LIN {X 0,Y 381.733,Z 858.539,A -85,B 0,C 180,E1 -11971.054,E2 -11971.054} C_VEL
LIN {X 0,Y 381.687,Z 857.929,A -85,B 0,C 180,E1 -11972.11,E2 -11972.11} C_VEL
LIN {X 0,Y 381.699,Z 855.51,A -85,B 0,C 180,E1 -11974.223,E2 -11974.223} C_VEL
LIN {X 0,Y 381.737,Z 852.426,A -85,B 0,C 180,E1 -11975.86,E2 -11975.86} C_VEL
LIN {X 0,Y 381.947,Z 848.497,A -85,B 0,C 180,E1 -11977.4,E2 -11977.4} C_VEL
LIN {X 0,Y 382.362,Z 842.256,A -85,B 0,C 180,E1 -11979.254,E2 -11979.254} C_VEL
LIN {X 0,Y 382.84,Z 835.448,A -85,B 0,C 180,E1 -11980.845,E2 -11980.845} C_VEL
LIN {X 0,Y 383.472,Z 828.515,A -85,B 0,C 180,E1 -11982.166,E2 -11982.166} C_VEL
LIN {X 0,Y 384.235,Z 820.166,A -85,B 0,C 180,E1 -11983.485,E2 -11983.485} C_VEL
LIN {X 0,Y 384.98,Z 811.335,A -85,B 0,C 180,E1 -11984.637,E2 -11984.637} C_VEL
LIN {X 0,Y 385.832,Z 801.143,A -85,B 0,C 180,E1 -11985.72,E2 -11985.72} C_VEL
LIN {X 0,Y 386.894,Z 788.721,A -85,B 0,C 180,E1 -11986.76,E2 -11986.76} C_VEL
LIN {X 0,Y 387.324,Z 779.513,A -85,B 0,C 180,E1 -11987.375,E2 -11987.375} C_VEL
LIN {X 0,Y 386.536,Z 767.148,A -85,B 0,C 180,E1 -11988.079,E2 -11988.079} C_VEL
LIN {X 0,Y 385.447,Z 753.763,A -85,B 0,C 180,E1 -11988.616,E2 -11988.616} C_VEL
LIN {X 0,Y 383.096,Z 737.702,A -85,B 0,C 180,E1 -11989.163,E2 -11989.163} C_VEL
LIN {X 0,Y 382.769,Z 734.559,A -85,B 0,C 180,E1 -11989.403,E2 -11989.403} C_VEL
LIN {X 0,Y 383.388,Z 721.586,A -85,B 0,C 180,E1 -11993.123,E2 -11993.123} C_VEL
LIN {X 0,Y 384.077,Z 710.72,A -85,B 0,C 180,E1 -11996.282,E2 -11996.282} C_VEL
LIN {X 0,Y 385.033,Z 697.753,A -85,B 0,C 180,E1 -12000.129,E2 -12000.129} C_VEL
LIN {X 0,Y 385.892,Z 687.901,A -85,B 0,C 180,E1 -12003.117,E2 -12003.117} C_VEL
LIN {X 0,Y 386.854,Z 678.017,A -85,B 0,C 180,E1 -12006.186,E2 -12006.186} C_VEL
LIN {X 0,Y 387.104,Z 673.941,A -85,B 0,C 180,E1 -12007.489,E2 -12007.489} C_VEL
LIN {X 0,Y 385.464,Z 664.856,A -85,B 0,C 180,E1 -12010.637,E2 -12010.637} C_VEL
LIN {X 0,Y 383.783,Z 656.694,A -85,B 0,C 180,E1 -12013.623,E2 -12013.623} C_VEL
LIN {X 0,Y 383.034,Z 652.774,A -85,B 0,C 180,E1 -12015.138,E2 -12015.138} C_VEL
LIN {X 0,Y 383.072,Z 652.769,A -85,B 0,C 180,E1 -12017.248,E2 -12017.248} C_VEL
LIN {X 0,Y 383.02,Z 652.776,A -85,B 0,C 180,E1 -12020.411,E2 -12020.411} C_VEL
LIN {X 0,Y 383.023,Z 652.777,A -85,B 0,C 180,E1 -12024.044,E2 -12024.044} C_VEL
LIN {X 0,Y 382.984,Z 652.778,A -85,B 0,C 180,E1 -12027.577,E2 -12027.577} C_VEL
LIN {X 0,Y 382.993,Z 652.776,A -85,B 0,C 180,E1 -12030.3,E2 -12030.3} C_VEL
LIN {X 0,Y 383.052,Z 652.77,A -85,B 0,C 180,E1 -12032.698,E2 -12032.698} C_VEL
LIN {X 0,Y 383.048,Z 652.767,A -85,B 0,C 180,E1 -12035.039,E2 -12035.039} C_VEL
LIN {X 0,Y 382.988,Z 652.778,A -85,B 0,C 180,E1 -12038.469,E2 -12038.469} C_VEL
LIN {X 0,Y 383.084,Z 652.764,A -85,B 0,C 180,E1 -12041.827,E2 -12041.827} C_VEL
LIN {X 0,Y 383.107,Z 652.762,A -85,B 0,C 180,E1 -12045.118,E2 -12045.118} C_VEL
LIN {X 0,Y 383.105,Z 652.765,A -85,B 0,C 180,E1 -12048.358,E2 -12048.358} C_VEL
LIN {X 0,Y 383.298,Z 652.741,A -85,B 0,C 180,E1 -12051.933,E2 -12051.933} C_VEL
LIN {X 0,Y 383.194,Z 652.754,A -85,B 0,C 180,E1 -12054.738,E2 -12054.738} C_VEL
LIN {X 0,Y 383.333,Z 652.738,A -85,B 0,C 180,E1 -12058.555,E2 -12058.555} C_VEL
LIN {X 0,Y 384.693,Z 658.546,A -85,B 0,C 180,E1 -12060.523,E2 -12060.523} C_VEL
LIN {X 0,Y 386.067,Z 666.754,A -85,B 0,C 180,E1 -12063.13,E2 -12063.13} C_VEL
LIN {X 0,Y 386.301,Z 673.618,A -85,B 0,C 180,E1 -12065.219,E2 -12065.219} C_VEL
LIN {X 0,Y 385.941,Z 682.388,A -85,B 0,C 180,E1 -12067.85,E2 -12067.85} C_VEL
LIN {X 0,Y 385.494,Z 692.988,A -85,B 0,C 180,E1 -12071.036,E2 -12071.036} C_VEL
LIN {X 0,Y 384.926,Z 705.565,A -85,B 0,C 180,E1 -12074.81,E2 -12074.81} C_VEL
LIN {X 0,Y 384.421,Z 716.408,A -85,B 0,C 180,E1 -12078.107,E2 -12078.107} C_VEL
LIN {X 0,Y 383.897,Z 728.338,A -85,B 0,C 180,E1 -12081.76,E2 -12081.76} C_VEL
LIN {X 0,Y 383.867,Z 728.923,A -85,B 0,C 180,E1 -12081.938,E2 -12081.938} C_VEL
LIN {X 0,Y 386.955,Z 743.243,A -85,B 0,C 180,E1 -12082.597,E2 -12082.597} C_VEL
LIN {X 0,Y 388.559,Z 754.403,A -85,B 0,C 180,E1 -12083.237,E2 -12083.237} C_VEL
LIN {X 0,Y 387.696,Z 767.572,A -85,B 0,C 180,E1 -12084.071,E2 -12084.071} C_VEL
LIN {X 0,Y 386.831,Z 778.255,A -85,B 0,C 180,E1 -12084.958,E2 -12084.958} C_VEL
LIN {X 0,Y 385.801,Z 789.749,A -85,B 0,C 180,E1 -12086.167,E2 -12086.167} C_VEL
LIN {X 0,Y 384.839,Z 799.637,A -85,B 0,C 180,E1 -12087.459,E2 -12087.459} C_VEL
LIN {X 0,Y 384.031,Z 807.845,A -85,B 0,C 180,E1 -12088.783,E2 -12088.783} C_VEL
LIN {X 0,Y 383.205,Z 816.257,A -85,B 0,C 180,E1 -12090.462,E2 -12090.462} C_VEL
LIN {X 0,Y 382.638,Z 823.079,A -85,B 0,C 180,E1 -12092.185,E2 -12092.185} C_VEL
LIN {X 0,Y 382.072,Z 828.954,A -85,B 0,C 180,E1 -12094.133,E2 -12094.133} C_VEL
LIN {X 0,Y 381.71,Z 833.209,A -85,B 0,C 180,E1 -12096.099,E2 -12096.099} C_VEL
LIN {X 0,Y 381.529,Z 835.452,A -85,B 0,C 180,E1 -12097.621,E2 -12097.621} C_VEL
LIN {X 0,Y 381.396,Z 836.916,A -85,B 0,C 180,E1 -12099.293,E2 -12099.293} C_VEL
LIN {X 0,Y 381.312,Z 837.371,A -85,B 0,C 180,E1 -12100.917,E2 -12100.917} C_VEL
LIN {X 0,Y 381.326,Z 836.543,A -85,B 0,C 180,E1 -12102.994,E2 -12102.994} C_VEL
LIN {X 0,Y 381.455,Z 835.07,A -85,B 0,C 180,E1 -12104.436,E2 -12104.436} C_VEL
LIN {X 0,Y 381.636,Z 832.771,A -85,B 0,C 180,E1 -12105.906,E2 -12105.906} C_VEL
LIN {X 0,Y 381.904,Z 829.532,A -85,B 0,C 180,E1 -12107.4,E2 -12107.4} C_VEL
LIN {X 0,Y 382.187,Z 825.206,A -85,B 0,C 180,E1 -12108.933,E2 -12108.933} C_VEL
LIN {X 0,Y 382.644,Z 819.682,A -85,B 0,C 180,E1 -12110.481,E2 -12110.481} C_VEL
LIN {X 0,Y 383.262,Z 812.689,A -85,B 0,C 180,E1 -12112.046,E2 -12112.046} C_VEL
LIN {X 0,Y 384.074,Z 803.926,A -85,B 0,C 180,E1 -12113.623,E2 -12113.623} C_VEL
LIN {X 0,Y 384.93,Z 794.235,A -85,B 0,C 180,E1 -12115.026,E2 -12115.026} C_VEL
LIN {X 0,Y 385.773,Z 783.871,A -85,B 0,C 180,E1 -12116.234,E2 -12116.234} C_VEL
LIN {X 0,Y 386.667,Z 772.826,A -85,B 0,C 180,E1 -12117.267,E2 -12117.267} C_VEL
LIN {X 0,Y 387.487,Z 761.215,A -85,B 0,C 180,E1 -12118.114,E2 -12118.114} C_VEL
LIN {X 0,Y 387.857,Z 753.357,A -85,B 0,C 180,E1 -12118.574,E2 -12118.574} C_VEL
LIN {X 0,Y 385.883,Z 740.488,A -85,B 0,C 180,E1 -12119.256,E2 -12119.256} C_VEL
LIN {X 0,Y 383.516,Z 728.322,A -85,B 0,C 180,E1 -12119.764,E2 -12119.764} C_VEL
LIN {X 0,Y 384.031,Z 718.573,A -85,B 0,C 180,E1 -12122.774,E2 -12122.774} C_VEL
LIN {X 0,Y 384.573,Z 707.203,A -85,B 0,C 180,E1 -12126.295,E2 -12126.295} C_VEL
LIN {X 0,Y 385.051,Z 696.202,A -85,B 0,C 180,E1 -12129.71,E2 -12129.71} C_VEL
LIN {X 0,Y 385.55,Z 685.478,A -85,B 0,C 180,E1 -12133.044,E2 -12133.044} C_VEL
LIN {X 0,Y 385.996,Z 675.003,A -85,B 0,C 180,E1 -12136.309,E2 -12136.309} C_VEL
LIN {X 0,Y 386.054,Z 669.909,A -85,B 0,C 180,E1 -12137.916,E2 -12137.916} C_VEL
LIN {X 0,Y 385.13,Z 662.906,A -85,B 0,C 180,E1 -12140.202,E2 -12140.202} C_VEL
LIN {X 0,Y 383.524,Z 654.044,A -85,B 0,C 180,E1 -12143.16,E2 -12143.16} C_VEL
LIN {X 0,Y 383.28,Z 652.747,A -85,B 0,C 180,E1 -12143.618,E2 -12143.618} C_VEL
LIN {X 0,Y 383.389,Z 652.732,A -85,B 0,C 180,E1 -12147.9,E2 -12147.9} C_VEL
LIN {X 0,Y 383.521,Z 652.714,A -85,B 0,C 180,E1 -12150.001,E2 -12150.001} C_VEL
LIN {X 0,Y 383.253,Z 652.747,A -85,B 0,C 180,E1 -12153.154,E2 -12153.154} C_VEL
LIN {X 0,Y 383.283,Z 652.739,A -85,B 0,C 180,E1 -12156.317,E2 -12156.317} C_VEL
LIN {X 0,Y 383.158,Z 652.755,A -85,B 0,C 180,E1 -12159.502,E2 -12159.502} C_VEL
LIN {X 0,Y 383.135,Z 652.761,A -85,B 0,C 180,E1 -12162.856,E2 -12162.856} C_VEL
LIN {X 0,Y 383.083,Z 652.768,A -85,B 0,C 180,E1 -12165.974,E2 -12165.974} C_VEL
LIN {X 0,Y 383.097,Z 652.767,A -85,B 0,C 180,E1 -12167.427,E2 -12167.427} C_VEL
LIN {X 0,Y 382.387,Z 652.857,A -85,B 0,C 180,E1 -12167.81,E2 -12167.81} C_VEL
LIN {X 0,Y 376.706,Z 653.565,A -85,B 0,C 180,E1 -12168.908,E2 -12168.908} C_VEL
LIN {X 0,Y 376.001,Z 653.65,A -85,B 0,C 180,E1 -12169.301,E2 -12169.301} C_VEL
LIN {X 0,Y 376.03,Z 653.649,A -85,B 0,C 180,E1 -12169.944,E2 -12169.944} C_VEL
LIN {X 0,Y 379.988,Z 666.978,A -85,B 0,C 180,E1 -12171.044,E2 -12171.044} C_VEL
LIN {X 0,Y 381.497,Z 672.992,A -85,B 0,C 180,E1 -12171.62,E2 -12171.62} C_VEL
LIN {X 0,Y 380.788,Z 683.919,A -85,B 0,C 180,E1 -12172.658,E2 -12172.658} C_VEL
LIN {X 0,Y 380.039,Z 694.118,A -85,B 0,C 180,E1 -12173.862,E2 -12173.862} C_VEL
LIN {X 0,Y 379.263,Z 703.439,A -85,B 0,C 180,E1 -12175.227,E2 -12175.227} C_VEL
LIN {X 0,Y 378.52,Z 711.615,A -85,B 0,C 180,E1 -12176.692,E2 -12176.692} C_VEL
LIN {X 0,Y 377.781,Z 718.994,A -85,B 0,C 180,E1 -12178.32,E2 -12178.32} C_VEL
LIN {X 0,Y 377.252,Z 724.681,A -85,B 0,C 180,E1 -12179.89,E2 -12179.89} C_VEL
LIN {X 0,Y 376.837,Z 729.243,A -85,B 0,C 180,E1 -12181.48,E2 -12181.48} C_VEL
LIN {X 0,Y 376.408,Z 733.369,A -85,B 0,C 180,E1 -12183.422,E2 -12183.422} C_VEL
LIN {X 0,Y 376.125,Z 736.147,A -85,B 0,C 180,E1 -12185.398,E2 -12185.398} C_VEL
LIN {X 0,Y 376.045,Z 737.235,A -85,B 0,C 180,E1 -12186.731,E2 -12186.731} C_VEL
LIN {X 0,Y 376.064,Z 737.75,A -85,B 0,C 180,E1 -12188.288,E2 -12188.288} C_VEL
LIN {X 0,Y 376.219,Z 737.339,A -85,B 0,C 180,E1 -12190.013,E2 -12190.013} C_VEL
LIN {X 0,Y 376.405,Z 735.988,A -85,B 0,C 180,E1 -12191.681,E2 -12191.681} C_VEL
LIN {X 0,Y 376.818,Z 733.11,A -85,B 0,C 180,E1 -12193.637,E2 -12193.637} C_VEL
LIN {X 0,Y 377.251,Z 730.106,A -85,B 0,C 180,E1 -12195.066,E2 -12195.066} C_VEL
LIN {X 0,Y 377.875,Z 725.016,A -85,B 0,C 180,E1 -12196.887,E2 -12196.887} C_VEL
LIN {X 0,Y 378.51,Z 719.748,A -85,B 0,C 180,E1 -12198.36,E2 -12198.36} C_VEL
LIN {X 0,Y 379.263,Z 713.164,A -85,B 0,C 180,E1 -12199.852,E2 -12199.852} C_VEL
LIN {X 0,Y 380.2,Z 704.709,A -85,B 0,C 180,E1 -12201.401,E2 -12201.401} C_VEL
LIN {X 0,Y 381.046,Z 696.501,A -85,B 0,C 180,E1 -12202.619,E2 -12202.619} C_VEL
LIN {X 0,Y 381.933,Z 685.637,A -85,B 0,C 180,E1 -12203.926,E2 -12203.926} C_VEL
LIN {X 0,Y 382.716,Z 675.004,A -85,B 0,C 180,E1 -12204.943,E2 -12204.943} C_VEL
LIN {X 0,Y 380.577,Z 667.189,A -85,B 0,C 180,E1 -12205.72,E2 -12205.72} C_VEL
LIN {X 0,Y 377.058,Z 656.704,A -85,B 0,C 180,E1 -12206.643,E2 -12206.643} C_VEL
LIN {X 0,Y 376.005,Z 653.65,A -85,B 0,C 180,E1 -12206.898,E2 -12206.898} C_VEL
LIN {X 0,Y 375.965,Z 653.658,A -85,B 0,C 180,E1 -12209.688,E2 -12209.688} C_VEL
LIN {X 0,Y 376.021,Z 653.643,A -85,B 0,C 180,E1 -12213.348,E2 -12213.348} C_VEL
LIN {X 0,Y 375.984,Z 653.643,A -85,B 0,C 180,E1 -12216.888,E2 -12216.888} C_VEL
LIN {X 0,Y 376.001,Z 653.649,A -85,B 0,C 180,E1 -12220.34,E2 -12220.34} C_VEL
LIN {X 0,Y 376.034,Z 653.647,A -85,B 0,C 180,E1 -12223.719,E2 -12223.719} C_VEL
LIN {X 0,Y 376.105,Z 653.635,A -85,B 0,C 180,E1 -12227.042,E2 -12227.042} C_VEL
LIN {X 0,Y 376.12,Z 653.634,A -85,B 0,C 180,E1 -12230.319,E2 -12230.319} C_VEL
LIN {X 0,Y 376.232,Z 653.612,A -85,B 0,C 180,E1 -12232.487,E2 -12232.487} C_VEL
LIN {X 0,Y 376.173,Z 653.625,A -85,B 0,C 180,E1 -12234.64,E2 -12234.64} C_VEL
LIN {X 0,Y 376.355,Z 653.6,A -85,B 0,C 180,E1 -12237.86,E2 -12237.86} C_VEL
LIN {X 0,Y 376.491,Z 653.584,A -85,B 0,C 180,E1 -12240,E2 -12240} C_VEL
LIN {X 0,Y 376.192,Z 653.622,A -85,B 0,C 180,E1 -12243.213,E2 -12243.213} C_VEL
LIN {X 0,Y 376.248,Z 653.619,A -85,B 0,C 180,E1 -12246.435,E2 -12246.435} C_VEL
LIN {X 0,Y 376.207,Z 653.616,A -85,B 0,C 180,E1 -12248.595,E2 -12248.595} C_VEL
LIN {X 0,Y 376.052,Z 653.643,A -85,B 0,C 180,E1 -12251.864,E2 -12251.864} C_VEL
LIN {X 0,Y 376.06,Z 653.639,A -85,B 0,C 180,E1 -12255.168,E2 -12255.168} C_VEL
LIN {X 0,Y 376.026,Z 653.646,A -85,B 0,C 180,E1 -12258.526,E2 -12258.526} C_VEL
LIN {X 0,Y 375.965,Z 653.653,A -85,B 0,C 180,E1 -12261.954,E2 -12261.954} C_VEL
LIN {X 0,Y 376.008,Z 653.644,A -85,B 0,C 180,E1 -12265.461,E2 -12265.461} C_VEL
LIN {X 0,Y 375.963,Z 653.654,A -85,B 0,C 180,E1 -12269.08,E2 -12269.08} C_VEL
LIN {X 0,Y 375.951,Z 653.655,A -85,B 0,C 180,E1 -12272.829,E2 -12272.829} C_VEL
LIN {X 0,Y 375.959,Z 653.656,A -85,B 0,C 180,E1 -12275.416,E2 -12275.416} C_VEL
LIN {X 0,Y 375.976,Z 653.654,A -85,B 0,C 180,E1 -12278.27,E2 -12278.27} C_VEL
LIN {X 0,Y 375.937,Z 653.659,A -85,B 0,C 180,E1 -12281.601,E2 -12281.601} C_VEL
LIN {X 0,Y 375.993,Z 653.819,A -85,B 0,C 180,E1 -12284.646,E2 -12284.646} C_VEL
LIN {X 0,Y 377.702,Z 662.116,A -85,B 0,C 180,E1 -12288.099,E2 -12288.099} C_VEL
LIN {X 0,Y 379.191,Z 669.985,A -85,B 0,C 180,E1 -12291.118,E2 -12291.118} C_VEL
LIN {X 0,Y 379.787,Z 674.451,A -85,B 0,C 180,E1 -12292.724,E2 -12292.724} C_VEL
LIN {X 0,Y 378.937,Z 683.037,A -85,B 0,C 180,E1 -12295.551,E2 -12295.551} C_VEL
LIN {X 0,Y 377.977,Z 693.317,A -85,B 0,C 180,E1 -12298.795,E2 -12298.795} C_VEL
LIN {X 0,Y 377.175,Z 704.555,A -85,B 0,C 180,E1 -12302.236,E2 -12302.236} C_VEL
LIN {X 0,Y 376.346,Z 717.964,A -85,B 0,C 180,E1 -12306.212,E2 -12306.212} C_VEL
LIN {X 0,Y 375.686,Z 732.397,A -85,B 0,C 180,E1 -12310.393,E2 -12310.393} C_VEL
LIN {X 0,Y 377.797,Z 748.756,A -85,B 0,C 180,E1 -12311.072,E2 -12311.072} C_VEL
LIN {X 0,Y 378.667,Z 760.461,A -85,B 0,C 180,E1 -12311.658,E2 -12311.658} C_VEL
LIN {X 0,Y 379.473,Z 773.4,A -85,B 0,C 180,E1 -12312.257,E2 -12312.257} C_VEL
LIN {X 0,Y 379.949,Z 782.049,A -85,B 0,C 180,E1 -12312.785,E2 -12312.785} C_VEL
LIN {X 0,Y 379.219,Z 793.186,A -85,B 0,C 180,E1 -12313.583,E2 -12313.583} C_VEL
LIN {X 0,Y 378.271,Z 804.709,A -85,B 0,C 180,E1 -12314.647,E2 -12314.647} C_VEL
LIN {X 0,Y 377.505,Z 814.451,A -85,B 0,C 180,E1 -12315.773,E2 -12315.773} C_VEL
LIN {X 0,Y 376.746,Z 823.602,A -85,B 0,C 180,E1 -12317.064,E2 -12317.064} C_VEL
LIN {X 0,Y 375.887,Z 832.783,A -85,B 0,C 180,E1 -12318.678,E2 -12318.678} C_VEL
LIN {X 0,Y 375.344,Z 840.149,A -85,B 0,C 180,E1 -12320.298,E2 -12320.298} C_VEL
LIN {X 0,Y 374.96,Z 846.031,A -85,B 0,C 180,E1 -12321.918,E2 -12321.918} C_VEL
LIN {X 0,Y 374.717,Z 851.111,A -85,B 0,C 180,E1 -12323.744,E2 -12323.744} C_VEL
LIN {X 0,Y 374.636,Z 854.998,A -85,B 0,C 180,E1 -12325.696,E2 -12325.696} C_VEL
LIN {X 0,Y 374.543,Z 856.529,A -85,B 0,C 180,E1 -12326.772,E2 -12326.772} C_VEL
LIN {X 0,Y 374.588,Z 857.595,A -85,B 0,C 180,E1 -12327.849,E2 -12327.849} C_VEL
LIN {X 0,Y 374.647,Z 858.252,A -85,B 0,C 180,E1 -12328.925,E2 -12328.925} C_VEL
LIN {X 0,Y 374.652,Z 858.511,A -85,B 0,C 180,E1 -12329.999,E2 -12329.999} C_VEL
LIN {X 0,Y 374.645,Z 858.351,A -85,B 0,C 180,E1 -12331.074,E2 -12331.074} C_VEL
LIN {X 0,Y 374.583,Z 857.749,A -85,B 0,C 180,E1 -12332.15,E2 -12332.15} C_VEL
LIN {X 0,Y 374.624,Z 855.347,A -85,B 0,C 180,E1 -12334.303,E2 -12334.303} C_VEL
LIN {X 0,Y 374.701,Z 851.678,A -85,B 0,C 180,E1 -12336.233,E2 -12336.233} C_VEL
LIN {X 0,Y 374.974,Z 846.745,A -85,B 0,C 180,E1 -12338.08,E2 -12338.08} C_VEL
LIN {X 0,Y 375.391,Z 841.125,A -85,B 0,C 180,E1 -12339.7,E2 -12339.7} C_VEL
LIN {X 0,Y 375.928,Z 834.099,A -85,B 0,C 180,E1 -12341.32,E2 -12341.32} C_VEL
LIN {X 0,Y 376.824,Z 825.308,A -85,B 0,C 180,E1 -12342.932,E2 -12342.932} C_VEL
LIN {X 0,Y 377.581,Z 816.47,A -85,B 0,C 180,E1 -12344.257,E2 -12344.257} C_VEL
LIN {X 0,Y 378.523,Z 806.455,A -85,B 0,C 180,E1 -12345.479,E2 -12345.479} C_VEL
LIN {X 0,Y 379.52,Z 795.532,A -85,B 0,C 180,E1 -12346.541,E2 -12346.541} C_VEL
LIN {X 0,Y 380.472,Z 783.686,A -85,B 0,C 180,E1 -12347.447,E2 -12347.447} C_VEL
LIN {X 0,Y 380.157,Z 774.532,A -85,B 0,C 180,E1 -12348.041,E2 -12348.041} C_VEL
LIN {X 0,Y 379.383,Z 761.031,A -85,B 0,C 180,E1 -12348.723,E2 -12348.723} C_VEL
LIN {X 0,Y 377.751,Z 746.489,A -85,B 0,C 180,E1 -12349.237,E2 -12349.237} C_VEL
LIN {X 0,Y 376.284,Z 738.142,A -85,B 0,C 180,E1 -12349.545,E2 -12349.545} C_VEL
LIN {X 0,Y 375.791,Z 732.903,A -85,B 0,C 180,E1 -12349.956,E2 -12349.956} C_VEL
LIN {X 0,Y 376.361,Z 720.97,A -85,B 0,C 180,E1 -12353.455,E2 -12353.455} C_VEL
LIN {X 0,Y 377.073,Z 710.511,A -85,B 0,C 180,E1 -12356.571,E2 -12356.571} C_VEL
LIN {X 0,Y 377.97,Z 698.756,A -85,B 0,C 180,E1 -12360.134,E2 -12360.134} C_VEL
LIN {X 0,Y 378.943,Z 688.125,A -85,B 0,C 180,E1 -12363.427,E2 -12363.427} C_VEL
LIN {X 0,Y 380.032,Z 677.442,A -85,B 0,C 180,E1 -12366.817,E2 -12366.817} C_VEL
LIN {X 0,Y 380.108,Z 675.081,A -85,B 0,C 180,E1 -12367.6,E2 -12367.6} C_VEL
LIN {X 0,Y 378.64,Z 666.825,A -85,B 0,C 180,E1 -12370.513,E2 -12370.513} C_VEL
LIN {X 0,Y 376.911,Z 658.484,A -85,B 0,C 180,E1 -12373.622,E2 -12373.622} C_VEL
LIN {X 0,Y 376.01,Z 653.649,A -85,B 0,C 180,E1 -12375.544,E2 -12375.544} C_VEL
LIN {X 0,Y 375.998,Z 653.649,A -85,B 0,C 180,E1 -12379.14,E2 -12379.14} C_VEL
LIN {X 0,Y 375.965,Z 653.651,A -85,B 0,C 180,E1 -12381.911,E2 -12381.911} C_VEL
LIN {X 0,Y 375.976,Z 653.646,A -85,B 0,C 180,E1 -12385.332,E2 -12385.332} C_VEL
LIN {X 0,Y 375.956,Z 653.649,A -85,B 0,C 180,E1 -12388.438,E2 -12388.438} C_VEL
LIN {X 0,Y 375.998,Z 653.648,A -85,B 0,C 180,E1 -12392.141,E2 -12392.141} C_VEL
LIN {X 0,Y 376.002,Z 653.643,A -85,B 0,C 180,E1 -12394.538,E2 -12394.538} C_VEL
LIN {X 0,Y 375.958,Z 653.655,A -85,B 0,C 180,E1 -12398.045,E2 -12398.045} C_VEL
LIN {X 0,Y 376.019,Z 653.647,A -85,B 0,C 180,E1 -12401.474,E2 -12401.474} C_VEL
LIN {X 0,Y 376.055,Z 653.64,A -85,B 0,C 180,E1 -12404.832,E2 -12404.832} C_VEL
LIN {X 0,Y 376.056,Z 653.642,A -85,B 0,C 180,E1 -12408.137,E2 -12408.137} C_VEL
LIN {X 0,Y 376.252,Z 653.619,A -85,B 0,C 180,E1 -12411.877,E2 -12411.877} C_VEL
LIN {X 0,Y 376.167,Z 653.629,A -85,B 0,C 180,E1 -12414.64,E2 -12414.64} C_VEL
LIN {X 0,Y 376.345,Z 653.711,A -85,B 0,C 180,E1 -12418.06,E2 -12418.06} C_VEL
LIN {X 0,Y 378.042,Z 661.077,A -85,B 0,C 180,E1 -12420.532,E2 -12420.532} C_VEL
LIN {X 0,Y 379.191,Z 667.571,A -85,B 0,C 180,E1 -12422.656,E2 -12422.656} C_VEL
LIN {X 0,Y 379.507,Z 674.423,A -85,B 0,C 180,E1 -12424.78,E2 -12424.78} C_VEL
LIN {X 0,Y 379.168,Z 683.23,A -85,B 0,C 180,E1 -12427.455,E2 -12427.455} C_VEL
LIN {X 0,Y 378.58,Z 695.681,A -85,B 0,C 180,E1 -12431.24,E2 -12431.24} C_VEL
LIN {X 0,Y 377.989,Z 707.324,A -85,B 0,C 180,E1 -12434.8,E2 -12434.8} C_VEL
LIN {X 0,Y 377.388,Z 719.19,A -85,B 0,C 180,E1 -12438.457,E2 -12438.457} C_VEL
LIN {X 0,Y 376.944,Z 729.185,A -85,B 0,C 180,E1 -12441.548,E2 -12441.548} C_VEL
LIN {X 0,Y 379.951,Z 742.477,A -85,B 0,C 180,E1 -12442.162,E2 -12442.162} C_VEL
LIN {X 0,Y 381.78,Z 754.505,A -85,B 0,C 180,E1 -12442.867,E2 -12442.867} C_VEL
LIN {X 0,Y 381.013,Z 767.435,A -85,B 0,C 180,E1 -12443.703,E2 -12443.703} C_VEL
LIN {X 0,Y 380.013,Z 779.218,A -85,B 0,C 180,E1 -12444.703,E2 -12444.703} C_VEL
LIN {X 0,Y 379.031,Z 789.726,A -85,B 0,C 180,E1 -12445.832,E2 -12445.832} C_VEL
LIN {X 0,Y 378.083,Z 798.539,A -85,B 0,C 180,E1 -12446.988,E2 -12446.988} C_VEL
LIN {X 0,Y 377.248,Z 807.146,A -85,B 0,C 180,E1 -12448.363,E2 -12448.363} C_VEL
LIN {X 0,Y 376.371,Z 815.256,A -85,B 0,C 180,E1 -12449.967,E2 -12449.967} C_VEL
LIN {X 0,Y 375.757,Z 821.813,A -85,B 0,C 180,E1 -12451.581,E2 -12451.581} C_VEL
LIN {X 0,Y 375.316,Z 826.164,A -85,B 0,C 180,E1 -12452.891,E2 -12452.891} C_VEL
LIN {X 0,Y 374.917,Z 830.276,A -85,B 0,C 180,E1 -12454.433,E2 -12454.433} C_VEL
LIN {X 0,Y 374.6,Z 833.811,A -85,B 0,C 180,E1 -12456.223,E2 -12456.223} C_VEL
LIN {X 0,Y 374.357,Z 836.427,A -85,B 0,C 180,E1 -12458.281,E2 -12458.281} C_VEL
LIN {X 0,Y 374.29,Z 837.309,A -85,B 0,C 180,E1 -12459.673,E2 -12459.673} C_VEL
LIN {X 0,Y 374.206,Z 837.512,A -85,B 0,C 180,E1 -12461.303,E2 -12461.303} C_VEL
LIN {X 0,Y 374.224,Z 836.81,A -85,B 0,C 180,E1 -12462.911,E2 -12462.911} C_VEL
LIN {X 0,Y 374.362,Z 835.238,A -85,B 0,C 180,E1 -12464.49,E2 -12464.49} C_VEL
LIN {X 0,Y 374.626,Z 831.804,A -85,B 0,C 180,E1 -12466.556,E2 -12466.556} C_VEL
LIN {X 0,Y 374.939,Z 828.152,A -85,B 0,C 180,E1 -12468.093,E2 -12468.093} C_VEL
LIN {X 0,Y 375.311,Z 823.5,A -85,B 0,C 180,E1 -12469.623,E2 -12469.623} C_VEL
LIN {X 0,Y 375.819,Z 817.737,A -85,B 0,C 180,E1 -12471.144,E2 -12471.144} C_VEL
LIN {X 0,Y 376.458,Z 810.734,A -85,B 0,C 180,E1 -12472.648,E2 -12472.648} C_VEL
LIN {X 0,Y 377.258,Z 802.586,A -85,B 0,C 180,E1 -12474.07,E2 -12474.07} C_VEL
LIN {X 0,Y 378.127,Z 792.733,A -85,B 0,C 180,E1 -12475.468,E2 -12475.468} C_VEL
LIN {X 0,Y 379.039,Z 782.436,A -85,B 0,C 180,E1 -12476.652,E2 -12476.652} C_VEL
LIN {X 0,Y 379.956,Z 770.606,A -85,B 0,C 180,E1 -12477.727,E2 -12477.727} C_VEL
LIN {X 0,Y 380.859,Z 758.198,A -85,B 0,C 180,E1 -12478.593,E2 -12478.593} C_VEL
LIN {X 0,Y 380.867,Z 753.147,A -85,B 0,C 180,E1 -12478.892,E2 -12478.892} C_VEL
LIN {X 0,Y 378.78,Z 740.113,A -85,B 0,C 180,E1 -12479.592,E2 -12479.592} C_VEL
LIN {X 0,Y 376.548,Z 728.448,A -85,B 0,C 180,E1 -12480.088,E2 -12480.088} C_VEL
LIN {X 0,Y 377.095,Z 717.676,A -85,B 0,C 180,E1 -12483.455,E2 -12483.455} C_VEL
LIN {X 0,Y 377.673,Z 706.375,A -85,B 0,C 180,E1 -12486.998,E2 -12486.998} C_VEL
LIN {X 0,Y 378.222,Z 695.319,A -85,B 0,C 180,E1 -12490.46,E2 -12490.46} C_VEL
LIN {X 0,Y 378.823,Z 682.845,A -85,B 0,C 180,E1 -12494.382,E2 -12494.382} C_VEL
LIN {X 0,Y 379.174,Z 672.388,A -85,B 0,C 180,E1 -12497.694,E2 -12497.694} C_VEL
LIN {X 0,Y 378.504,Z 666.076,A -85,B 0,C 180,E1 -12499.767,E2 -12499.767} C_VEL
LIN {X 0,Y 376.79,Z 656.38,A -85,B 0,C 180,E1 -12503.037,E2 -12503.037} C_VEL
LIN {X 0,Y 376.225,Z 653.627,A -85,B 0,C 180,E1 -12504.036,E2 -12504.036} C_VEL
LIN {X 0,Y 376.355,Z 653.608,A -85,B 0,C 180,E1 -12507.86,E2 -12507.86} C_VEL
LIN {X 0,Y 376.49,Z 653.59,A -85,B 0,C 180,E1 -12510.001,E2 -12510.001} C_VEL
LIN {X 0,Y 376.191,Z 653.626,A -85,B 0,C 180,E1 -12513.213,E2 -12513.213} C_VEL
LIN {X 0,Y 376.241,Z 653.616,A -85,B 0,C 180,E1 -12516.436,E2 -12516.436} C_VEL
LIN {X 0,Y 376.125,Z 653.63,A -85,B 0,C 180,E1 -12519.682,E2 -12519.682} C_VEL
LIN {X 0,Y 376.091,Z 653.639,A -85,B 0,C 180,E1 -12523.658,E2 -12523.658} C_VEL
LIN {X 0,Y 376.046,Z 653.646,A -85,B 0,C 180,E1 -12527.608,E2 -12527.608} C_VEL
LIN {X 0,Y 376.001,Z 653.65,A -85,B 0,C 180,E1 -12529.301,E2 -12529.301} C_VEL
LIN {X 0,Y 375.989,Z 654.402,A -85,B 0,C 180,E1 -12529.661,E2 -12529.661} C_VEL
LIN {X 0,Y 375.944,Z 656.577,A -85,B 0,C 180,E1 -12530.015,E2 -12530.015} C_VEL
LIN {X 0,Y 375.855,Z 660.662,A -85,B 0,C 180,E1 -12530.376,E2 -12530.376} C_VEL
LIN {X 0,Y 374.837,Z 674.39,A -85,B 0,C 180,E1 -12531.373,E2 -12531.373} C_VEL
LIN {X 0,Y 374.265,Z 680.346,A -85,B 0,C 180,E1 -12531.934,E2 -12531.934} C_VEL
LIN {X 0,Y 373.485,Z 691.243,A -85,B 0,C 180,E1 -12533.137,E2 -12533.137} C_VEL
LIN {X 0,Y 372.659,Z 701.228,A -85,B 0,C 180,E1 -12534.513,E2 -12534.513} C_VEL
LIN {X 0,Y 371.821,Z 710.383,A -85,B 0,C 180,E1 -12536.07,E2 -12536.07} C_VEL
LIN {X 0,Y 371.028,Z 717.92,A -85,B 0,C 180,E1 -12537.665,E2 -12537.665} C_VEL
LIN {X 0,Y 370.347,Z 725.004,A -85,B 0,C 180,E1 -12539.565,E2 -12539.565} C_VEL
LIN {X 0,Y 369.792,Z 730.841,A -85,B 0,C 180,E1 -12541.641,E2 -12541.641} C_VEL
LIN {X 0,Y 369.384,Z 734.589,A -85,B 0,C 180,E1 -12543.488,E2 -12543.488} C_VEL
LIN {X 0,Y 369.129,Z 736.801,A -85,B 0,C 180,E1 -12545.046,E2 -12545.046} C_VEL
LIN {X 0,Y 369.012,Z 738.335,A -85,B 0,C 180,E1 -12546.879,E2 -12546.879} C_VEL
LIN {X 0,Y 369.087,Z 738.75,A -85,B 0,C 180,E1 -12548.931,E2 -12548.931} C_VEL
LIN {X 0,Y 369.236,Z 738.167,A -85,B 0,C 180,E1 -12550.416,E2 -12550.416} C_VEL
LIN {X 0,Y 369.455,Z 736.638,A -85,B 0,C 180,E1 -12552.108,E2 -12552.108} C_VEL
LIN {X 0,Y 369.86,Z 734.153,A -85,B 0,C 180,E1 -12553.775,E2 -12553.775} C_VEL
LIN {X 0,Y 370.374,Z 730.722,A -85,B 0,C 180,E1 -12555.405,E2 -12555.405} C_VEL
LIN {X 0,Y 370.956,Z 726.338,A -85,B 0,C 180,E1 -12556.997,E2 -12556.997} C_VEL
LIN {X 0,Y 371.74,Z 720.205,A -85,B 0,C 180,E1 -12558.736,E2 -12558.736} C_VEL
LIN {X 0,Y 372.549,Z 713.448,A -85,B 0,C 180,E1 -12560.264,E2 -12560.264} C_VEL
LIN {X 0,Y 373.495,Z 705.17,A -85,B 0,C 180,E1 -12561.775,E2 -12561.775} C_VEL
LIN {X 0,Y 374.43,Z 696.313,A -85,B 0,C 180,E1 -12563.085,E2 -12563.085} C_VEL
LIN {X 0,Y 375.388,Z 685.431,A -85,B 0,C 180,E1 -12564.387,E2 -12564.387} C_VEL
LIN {X 0,Y 376.04,Z 676.505,A -85,B 0,C 180,E1 -12565.249,E2 -12565.249} C_VEL
LIN {X 0,Y 373.212,Z 666.683,A -85,B 0,C 180,E1 -12566.254,E2 -12566.254} C_VEL
LIN {X 0,Y 369.027,Z 655.114,A -85,B 0,C 180,E1 -12567.279,E2 -12567.279} C_VEL
LIN {X 0,Y 368.919,Z 654.536,A -85,B 0,C 180,E1 -12567.358,E2 -12567.358} C_VEL
LIN {X 0,Y 368.916,Z 654.53,A -85,B 0,C 180,E1 -12570.31,E2 -12570.31} C_VEL
LIN {X 0,Y 369.001,Z 654.517,A -85,B 0,C 180,E1 -12574.02,E2 -12574.02} C_VEL
LIN {X 0,Y 368.926,Z 654.523,A -85,B 0,C 180,E1 -12577.605,E2 -12577.605} C_VEL
LIN {X 0,Y 368.985,Z 654.523,A -85,B 0,C 180,E1 -12581.107,E2 -12581.107} C_VEL
LIN {X 0,Y 369.002,Z 654.521,A -85,B 0,C 180,E1 -12584.536,E2 -12584.536} C_VEL
LIN {X 0,Y 369.007,Z 654.52,A -85,B 0,C 180,E1 -12587.907,E2 -12587.907} C_VEL
LIN {X 0,Y 369.231,Z 654.488,A -85,B 0,C 180,E1 -12591.801,E2 -12591.801} C_VEL
LIN {X 0,Y 369.146,Z 654.501,A -85,B 0,C 180,E1 -12594.538,E2 -12594.538} C_VEL
LIN {X 0,Y 369.32,Z 654.476,A -85,B 0,C 180,E1 -12597.819,E2 -12597.819} C_VEL
LIN {X 0,Y 369.46,Z 654.459,A -85,B 0,C 180,E1 -12600,E2 -12600} C_VEL
LIN {X 0,Y 369.321,Z 654.478,A -85,B 0,C 180,E1 -12602.181,E2 -12602.181} C_VEL
LIN {X 0,Y 369.21,Z 654.495,A -85,B 0,C 180,E1 -12606.558,E2 -12606.558} C_VEL
LIN {X 0,Y 369.139,Z 654.495,A -85,B 0,C 180,E1 -12608.761,E2 -12608.761} C_VEL
LIN {X 0,Y 369.007,Z 654.518,A -85,B 0,C 180,E1 -12612.093,E2 -12612.093} C_VEL
LIN {X 0,Y 369,Z 654.519,A -85,B 0,C 180,E1 -12615.465,E2 -12615.465} C_VEL
LIN {X 0,Y 368.984,Z 654.519,A -85,B 0,C 180,E1 -12618.893,E2 -12618.893} C_VEL
LIN {X 0,Y 368.934,Z 654.527,A -85,B 0,C 180,E1 -12622.395,E2 -12622.395} C_VEL
LIN {X 0,Y 369.002,Z 654.517,A -85,B 0,C 180,E1 -12625.98,E2 -12625.98} C_VEL
LIN {X 0,Y 368.917,Z 654.531,A -85,B 0,C 180,E1 -12629.69,E2 -12629.69} C_VEL
LIN {X 0,Y 368.899,Z 654.534,A -85,B 0,C 180,E1 -12633.043,E2 -12633.043} C_VEL
LIN {X 0,Y 368.919,Z 654.534,A -85,B 0,C 180,E1 -12636.197,E2 -12636.197} C_VEL
LIN {X 0,Y 368.905,Z 654.538,A -85,B 0,C 180,E1 -12638.953,E2 -12638.953} C_VEL
LIN {X 0,Y 368.884,Z 654.538,A -85,B 0,C 180,E1 -12642.009,E2 -12642.009} C_VEL
LIN {X 0,Y 368.961,Z 654.72,A -85,B 0,C 180,E1 -12644.161,E2 -12644.161} C_VEL
LIN {X 0,Y 370.648,Z 662.896,A -85,B 0,C 180,E1 -12647.689,E2 -12647.689} C_VEL
LIN {X 0,Y 372.117,Z 670.664,A -85,B 0,C 180,E1 -12650.746,E2 -12650.746} C_VEL
LIN {X 0,Y 372.839,Z 674.953,A -85,B 0,C 180,E1 -12652.345,E2 -12652.345} C_VEL
LIN {X 0,Y 372.147,Z 682.37,A -85,B 0,C 180,E1 -12654.866,E2 -12654.866} C_VEL
LIN {X 0,Y 371.056,Z 693.476,A -85,B 0,C 180,E1 -12658.466,E2 -12658.466} C_VEL
LIN {X 0,Y 370.114,Z 705.643,A -85,B 0,C 180,E1 -12662.275,E2 -12662.275} C_VEL
LIN {X 0,Y 369.291,Z 717.871,A -85,B 0,C 180,E1 -12665.993,E2 -12665.993} C_VEL
LIN {X 0,Y 368.643,Z 731.327,A -85,B 0,C 180,E1 -12669.985,E2 -12669.985} C_VEL
LIN {X 0,Y 370.67,Z 745.925,A -85,B 0,C 180,E1 -12670.586,E2 -12670.586} C_VEL
LIN {X 0,Y 371.895,Z 761.548,A -85,B 0,C 180,E1 -12671.39,E2 -12671.39} C_VEL
LIN {X 0,Y 372.607,Z 774.142,A -85,B 0,C 180,E1 -12672.006,E2 -12672.006} C_VEL
LIN {X 0,Y 373.068,Z 782.405,A -85,B 0,C 180,E1 -12672.528,E2 -12672.528} C_VEL
LIN {X 0,Y 372.229,Z 794.163,A -85,B 0,C 180,E1 -12673.406,E2 -12673.406} C_VEL
LIN {X 0,Y 371.274,Z 805.466,A -85,B 0,C 180,E1 -12674.491,E2 -12674.491} C_VEL
LIN {X 0,Y 370.45,Z 815.683,A -85,B 0,C 180,E1 -12675.721,E2 -12675.721} C_VEL
LIN {X 0,Y 369.639,Z 824.856,A -85,B 0,C 180,E1 -12677.09,E2 -12677.09} C_VEL
LIN {X 0,Y 368.769,Z 833.771,A -85,B 0,C 180,E1 -12678.735,E2 -12678.735} C_VEL
LIN {X 0,Y 368.222,Z 840.906,A -85,B 0,C 180,E1 -12680.386,E2 -12680.386} C_VEL
LIN {X 0,Y 367.907,Z 845.72,A -85,B 0,C 180,E1 -12681.762,E2 -12681.762} C_VEL
LIN {X 0,Y 367.65,Z 850.348,A -85,B 0,C 180,E1 -12683.413,E2 -12683.413} C_VEL
LIN {X 0,Y 367.581,Z 852.772,A -85,B 0,C 180,E1 -12684.514,E2 -12684.514} C_VEL
LIN {X 0,Y 367.562,Z 854.746,A -85,B 0,C 180,E1 -12685.613,E2 -12685.613} C_VEL
LIN {X 0,Y 367.458,Z 856.29,A -85,B 0,C 180,E1 -12686.71,E2 -12686.71} C_VEL
LIN {X 0,Y 367.486,Z 857.371,A -85,B 0,C 180,E1 -12687.807,E2 -12687.807} C_VEL
LIN {X 0,Y 367.561,Z 858.038,A -85,B 0,C 180,E1 -12688.904,E2 -12688.904} C_VEL
LIN {X 0,Y 367.584,Z 858.307,A -85,B 0,C 180,E1 -12689.999,E2 -12689.999} C_VEL
LIN {X 0,Y 367.544,Z 858.162,A -85,B 0,C 180,E1 -12691.095,E2 -12691.095} C_VEL
LIN {X 0,Y 367.48,Z 857.569,A -85,B 0,C 180,E1 -12692.191,E2 -12692.191} C_VEL
LIN {X 0,Y 367.55,Z 855.183,A -85,B 0,C 180,E1 -12694.386,E2 -12694.386} C_VEL
LIN {X 0,Y 367.595,Z 851.929,A -85,B 0,C 180,E1 -12696.182,E2 -12696.182} C_VEL
LIN {X 0,Y 367.915,Z 846.623,A -85,B 0,C 180,E1 -12698.236,E2 -12698.236} C_VEL
LIN {X 0,Y 368.368,Z 841.034,A -85,B 0,C 180,E1 -12699.887,E2 -12699.887} C_VEL
LIN {X 0,Y 368.942,Z 834.056,A -85,B 0,C 180,E1 -12701.537,E2 -12701.537} C_VEL
LIN {X 0,Y 369.896,Z 825.317,A -85,B 0,C 180,E1 -12703.179,E2 -12703.179} C_VEL
LIN {X 0,Y 370.826,Z 815.4,A -85,B 0,C 180,E1 -12704.684,E2 -12704.684} C_VEL
LIN {X 0,Y 371.803,Z 805.324,A -85,B 0,C 180,E1 -12705.907,E2 -12705.907} C_VEL
LIN {X 0,Y 372.889,Z 794.2,A -85,B 0,C 180,E1 -12706.985,E2 -12706.985} C_VEL
LIN {X 0,Y 373.812,Z 782.163,A -85,B 0,C 180,E1 -12707.904,E2 -12707.904} C_VEL
LIN {X 0,Y 373.159,Z 769.293,A -85,B 0,C 180,E1 -12708.708,E2 -12708.708} C_VEL
LIN {X 0,Y 372.202,Z 755.761,A -85,B 0,C 180,E1 -12709.33,E2 -12709.33} C_VEL
LIN {X 0,Y 370.078,Z 741.082,A -85,B 0,C 180,E1 -12709.844,E2 -12709.844} C_VEL
LIN {X 0,Y 369.507,Z 738.139,A -85,B 0,C 180,E1 -12709.967,E2 -12709.967} C_VEL
LIN {X 0,Y 368.754,Z 731.278,A -85,B 0,C 180,E1 -12710.514,E2 -12710.514} C_VEL
LIN {X 0,Y 369.395,Z 719.542,A -85,B 0,C 180,E1 -12714.043,E2 -12714.043} C_VEL
LIN {X 0,Y 370.267,Z 707.555,A -85,B 0,C 180,E1 -12717.711,E2 -12717.711} C_VEL
LIN {X 0,Y 371.348,Z 695.055,A -85,B 0,C 180,E1 -12721.608,E2 -12721.608} C_VEL
LIN {X 0,Y 372.475,Z 684.022,A -85,B 0,C 180,E1 -12725.133,E2 -12725.133} C_VEL
LIN {X 0,Y 373.078,Z 678.1,A -85,B 0,C 180,E1 -12727.07,E2 -12727.07} C_VEL
LIN {X 0,Y 372.796,Z 674.06,A -85,B 0,C 180,E1 -12728.47,E2 -12728.47} C_VEL
LIN {X 0,Y 370.991,Z 664.64,A -85,B 0,C 180,E1 -12731.92,E2 -12731.92} C_VEL
LIN {X 0,Y 368.955,Z 654.528,A -85,B 0,C 180,E1 -12735.91,E2 -12735.91} C_VEL
LIN {X 0,Y 368.95,Z 654.527,A -85,B 0,C 180,E1 -12739.635,E2 -12739.635} C_VEL
LIN {X 0,Y 368.9,Z 654.531,A -85,B 0,C 180,E1 -12743.143,E2 -12743.143} C_VEL
LIN {X 0,Y 368.893,Z 654.535,A -85,B 0,C 180,E1 -12746.461,E2 -12746.461} C_VEL
LIN {X 0,Y 368.919,Z 654.529,A -85,B 0,C 180,E1 -12750.31,E2 -12750.31} C_VEL
LIN {X 0,Y 368.977,Z 654.522,A -85,B 0,C 180,E1 -12753.534,E2 -12753.534} C_VEL
LIN {X 0,Y 368.962,Z 654.524,A -85,B 0,C 180,E1 -12756.421,E2 -12756.421} C_VEL
LIN {X 0,Y 368.931,Z 654.525,A -85,B 0,C 180,E1 -12759.947,E2 -12759.947} C_VEL
LIN {X 0,Y 368.972,Z 654.526,A -85,B 0,C 180,E1 -12763.398,E2 -12763.398} C_VEL
LIN {X 0,Y 369.055,Z 654.513,A -85,B 0,C 180,E1 -12766.79,E2 -12766.79} C_VEL
LIN {X 0,Y 369.068,Z 654.513,A -85,B 0,C 180,E1 -12770.132,E2 -12770.132} C_VEL
LIN {X 0,Y 369.183,Z 654.5,A -85,B 0,C 180,E1 -12772.342,E2 -12772.342} C_VEL
LIN {X 0,Y 369.139,Z 654.504,A -85,B 0,C 180,E1 -12774.537,E2 -12774.537} C_VEL
LIN {X 0,Y 369.235,Z 654.598,A -85,B 0,C 180,E1 -12777.409,E2 -12777.409} C_VEL
LIN {X 0,Y 371.138,Z 662.036,A -85,B 0,C 180,E1 -12780,E2 -12780} C_VEL
LIN {X 0,Y 372.508,Z 670.172,A -85,B 0,C 180,E1 -12782.703,E2 -12782.703} C_VEL
LIN {X 0,Y 372.71,Z 677.026,A -85,B 0,C 180,E1 -12784.867,E2 -12784.867} C_VEL
LIN {X 0,Y 372.29,Z 685.832,A -85,B 0,C 180,E1 -12787.593,E2 -12787.593} C_VEL
LIN {X 0,Y 371.636,Z 698.24,A -85,B 0,C 180,E1 -12791.453,E2 -12791.453} C_VEL
LIN {X 0,Y 371.09,Z 708.999,A -85,B 0,C 180,E1 -12794.751,E2 -12794.751} C_VEL
LIN {X 0,Y 370.434,Z 720.85,A -85,B 0,C 180,E1 -12798.45,E2 -12798.45} C_VEL
LIN {X 0,Y 370.039,Z 729.492,A -85,B 0,C 180,E1 -12801.116,E2 -12801.116} C_VEL
LIN {X 0,Y 373.164,Z 743.028,A -85,B 0,C 180,E1 -12801.773,E2 -12801.773} C_VEL
LIN {X 0,Y 375.126,Z 755.9,A -85,B 0,C 180,E1 -12802.568,E2 -12802.568} C_VEL
LIN {X 0,Y 374.286,Z 767.96,A -85,B 0,C 180,E1 -12803.37,E2 -12803.37} C_VEL
LIN {X 0,Y 373.302,Z 778.987,A -85,B 0,C 180,E1 -12804.32,E2 -12804.32} C_VEL
LIN {X 0,Y 372.187,Z 790.37,A -85,B 0,C 180,E1 -12805.564,E2 -12805.564} C_VEL
LIN {X 0,Y 371.104,Z 800.074,A -85,B 0,C 180,E1 -12806.881,E2 -12806.881} C_VEL
LIN {X 0,Y 370.204,Z 808.677,A -85,B 0,C 180,E1 -12808.333,E2 -12808.333} C_VEL
LIN {X 0,Y 369.297,Z 816.563,A -85,B 0,C 180,E1 -12809.971,E2 -12809.971} C_VEL
LIN {X 0,Y 368.681,Z 822.918,A -85,B 0,C 180,E1 -12811.615,E2 -12811.615} C_VEL
LIN {X 0,Y 368.042,Z 828.903,A -85,B 0,C 180,E1 -12813.626,E2 -12813.626} C_VEL
LIN {X 0,Y 367.614,Z 833.31,A -85,B 0,C 180,E1 -12815.668,E2 -12815.668} C_VEL
LIN {X 0,Y 367.318,Z 836.187,A -85,B 0,C 180,E1 -12817.753,E2 -12817.753} C_VEL
LIN {X 0,Y 367.2,Z 837.323,A -85,B 0,C 180,E1 -12819.168,E2 -12819.168} C_VEL
LIN {X 0,Y 367.146,Z 837.747,A -85,B 0,C 180,E1 -12820.605,E2 -12820.605} C_VEL
LIN {X 0,Y 367.097,Z 837.484,A -85,B 0,C 180,E1 -12822.072,E2 -12822.072} C_VEL
LIN {X 0,Y 367.173,Z 836.502,A -85,B 0,C 180,E1 -12823.556,E2 -12823.556} C_VEL
LIN {X 0,Y 367.331,Z 834.717,A -85,B 0,C 180,E1 -12825.065,E2 -12825.065} C_VEL
LIN {X 0,Y 367.563,Z 832.052,A -85,B 0,C 180,E1 -12826.6,E2 -12826.6} C_VEL
LIN {X 0,Y 367.863,Z 828.416,A -85,B 0,C 180,E1 -12828.167,E2 -12828.167} C_VEL
LIN {X 0,Y 368.318,Z 822.63,A -85,B 0,C 180,E1 -12830.07,E2 -12830.07} C_VEL
LIN {X 0,Y 369.052,Z 815.218,A -85,B 0,C 180,E1 -12831.929,E2 -12831.929} C_VEL
LIN {X 0,Y 369.76,Z 807.518,A -85,B 0,C 180,E1 -12833.475,E2 -12833.475} C_VEL
LIN {X 0,Y 370.727,Z 797.963,A -85,B 0,C 180,E1 -12835.013,E2 -12835.013} C_VEL
LIN {X 0,Y 371.757,Z 787.316,A -85,B 0,C 180,E1 -12836.392,E2 -12836.392} C_VEL
LIN {X 0,Y 372.58,Z 777.513,A -85,B 0,C 180,E1 -12837.418,E2 -12837.418} C_VEL
LIN {X 0,Y 373.53,Z 766.037,A -85,B 0,C 180,E1 -12838.368,E2 -12838.368} C_VEL
LIN {X 0,Y 374.158,Z 755.494,A -85,B 0,C 180,E1 -12839.057,E2 -12839.057} C_VEL
LIN {X 0,Y 372.179,Z 742.34,A -85,B 0,C 180,E1 -12839.817,E2 -12839.817} C_VEL
LIN {X 0,Y 369.571,Z 728.62,A -85,B 0,C 180,E1 -12840.414,E2 -12840.414} C_VEL
LIN {X 0,Y 370.238,Z 716.897,A -85,B 0,C 180,E1 -12844.114,E2 -12844.114} C_VEL
LIN {X 0,Y 370.819,Z 705.471,A -85,B 0,C 180,E1 -12847.726,E2 -12847.726} C_VEL
LIN {X 0,Y 371.358,Z 694.429,A -85,B 0,C 180,E1 -12851.233,E2 -12851.233} C_VEL
LIN {X 0,Y 371.914,Z 683.655,A -85,B 0,C 180,E1 -12854.66,E2 -12854.66} C_VEL
LIN {X 0,Y 372.264,Z 674.872,A -85,B 0,C 180,E1 -12857.461,E2 -12857.461} C_VEL
LIN {X 0,Y 371.823,Z 669.069,A -85,B 0,C 180,E1 -12859.381,E2 -12859.381} C_VEL
LIN {X 0,Y 370.346,Z 660.301,A -85,B 0,C 180,E1 -12862.367,E2 -12862.367} C_VEL
LIN {X 0,Y 369.155,Z 654.506,A -85,B 0,C 180,E1 -12864.401,E2 -12864.401} C_VEL
LIN {X 0,Y 369.32,Z 654.484,A -85,B 0,C 180,E1 -12867.819,E2 -12867.819} C_VEL
LIN {X 0,Y 369.46,Z 654.466,A -85,B 0,C 180,E1 -12870.001,E2 -12870.001} C_VEL
LIN {X 0,Y 369.32,Z 654.482,A -85,B 0,C 180,E1 -12872.182,E2 -12872.182} C_VEL
LIN {X 0,Y 369.201,Z 654.492,A -85,B 0,C 180,E1 -12876.559,E2 -12876.559} C_VEL
LIN {X 0,Y 369.124,Z 654.506,A -85,B 0,C 180,E1 -12878.762,E2 -12878.762} C_VEL
LIN {X 0,Y 369.015,Z 654.52,A -85,B 0,C 180,E1 -12882.093,E2 -12882.093} C_VEL
LIN {X 0,Y 369.001,Z 654.523,A -85,B 0,C 180,E1 -12885.465,E2 -12885.465} C_VEL
LIN {X 0,Y 368.989,Z 654.526,A -85,B 0,C 180,E1 -12888.893,E2 -12888.893} C_VEL
LIN {X 0,Y 368.983,Z 654.527,A -85,B 0,C 180,E1 -12889.616,E2 -12889.616} C_VEL
LIN {X 0,Y 372.877,Z 667.349,A -85,B 0,C 180,E1 -12890.696,E2 -12890.696} C_VEL
LIN {X 0,Y 374.578,Z 673.688,A -85,B 0,C 180,E1 -12891.317,E2 -12891.317} C_VEL
LIN {X 0,Y 374.265,Z 680.346,A -85,B 0,C 180,E1 -12891.934,E2 -12891.934} C_VEL
LIN {X 0,Y 373.287,Z 685.284,A -85,B 0,C 180,E1 -12892.409,E2 -12892.409} C_VEL
LIN {X 0,Y 369.959,Z 693.125,A -85,B 0,C 180,E1 -12893.193,E2 -12893.193} C_VEL
LIN {X 0,Y 366.595,Z 700.564,A -85,B 0,C 180,E1 -12894.072,E2 -12894.072} C_VEL
LIN {X 0,Y 365.558,Z 704.756,A -85,B 0,C 180,E1 -12894.698,E2 -12894.698} C_VEL
LIN {X 0,Y 364.674,Z 713.531,A -85,B 0,C 180,E1 -12896.312,E2 -12896.312} C_VEL
LIN {X 0,Y 363.921,Z 720.626,A -85,B 0,C 180,E1 -12897.925,E2 -12897.925} C_VEL
LIN {X 0,Y 363.256,Z 727.146,A -85,B 0,C 180,E1 -12899.798,E2 -12899.798} C_VEL
LIN {X 0,Y 362.812,Z 731.808,A -85,B 0,C 180,E1 -12901.535,E2 -12901.535} C_VEL
LIN {X 0,Y 362.353,Z 735.694,A -85,B 0,C 180,E1 -12903.488,E2 -12903.488} C_VEL
LIN {X 0,Y 362.071,Z 738.453,A -85,B 0,C 180,E1 -12905.614,E2 -12905.614} C_VEL
LIN {X 0,Y 361.994,Z 739.549,A -85,B 0,C 180,E1 -12907.25,E2 -12907.25} C_VEL
LIN {X 0,Y 362.073,Z 739.781,A -85,B 0,C 180,E1 -12909.066,E2 -12909.066} C_VEL
LIN {X 0,Y 362.324,Z 738.646,A -85,B 0,C 180,E1 -12911.262,E2 -12911.262} C_VEL
LIN {X 0,Y 362.783,Z 735.999,A -85,B 0,C 180,E1 -12913.45,E2 -12913.45} C_VEL
LIN {X 0,Y 363.216,Z 733.234,A -85,B 0,C 180,E1 -12914.93,E2 -12914.93} C_VEL
LIN {X 0,Y 363.923,Z 728.498,A -85,B 0,C 180,E1 -12916.834,E2 -12916.834} C_VEL
LIN {X 0,Y 364.756,Z 722.249,A -85,B 0,C 180,E1 -12918.716,E2 -12918.716} C_VEL
LIN {X 0,Y 365.588,Z 715.773,A -85,B 0,C 180,E1 -12920.26,E2 -12920.26} C_VEL
LIN {X 0,Y 366.665,Z 706.975,A -85,B 0,C 180,E1 -12921.948,E2 -12921.948} C_VEL
LIN {X 0,Y 367.715,Z 697.475,A -85,B 0,C 180,E1 -12923.392,E2 -12923.392} C_VEL
LIN {X 0,Y 368.636,Z 687.645,A -85,B 0,C 180,E1 -12924.602,E2 -12924.602} C_VEL
LIN {X 0,Y 369.339,Z 678.515,A -85,B 0,C 180,E1 -12925.521,E2 -12925.521} C_VEL
LIN {X 0,Y 366.709,Z 669.043,A -85,B 0,C 180,E1 -12926.527,E2 -12926.527} C_VEL
LIN {X 0,Y 362.991,Z 658.714,A -85,B 0,C 180,E1 -12927.502,E2 -12927.502} C_VEL
LIN {X 0,Y 361.87,Z 655.411,A -85,B 0,C 180,E1 -12927.8,E2 -12927.8} C_VEL
LIN {X 0,Y 361.901,Z 655.402,A -85,B 0,C 180,E1 -12930.955,E2 -12930.955} C_VEL
LIN {X 0,Y 361.955,Z 655.394,A -85,B 0,C 180,E1 -12933.475,E2 -12933.475} C_VEL
LIN {X 0,Y 361.883,Z 655.398,A -85,B 0,C 180,E1 -12937.144,E2 -12937.144} C_VEL
LIN {X 0,Y 361.923,Z 655.402,A -85,B 0,C 180,E1 -12940.724,E2 -12940.724} C_VEL
LIN {X 0,Y 361.95,Z 655.402,A -85,B 0,C 180,E1 -12944.226,E2 -12944.226} C_VEL
LIN {X 0,Y 362,Z 655.393,A -85,B 0,C 180,E1 -12946.528,E2 -12946.528} C_VEL
LIN {X 0,Y 362.033,Z 655.39,A -85,B 0,C 180,E1 -12949.938,E2 -12949.938} C_VEL
LIN {X 0,Y 362.153,Z 655.366,A -85,B 0,C 180,E1 -12952.193,E2 -12952.193} C_VEL
LIN {X 0,Y 362.12,Z 655.377,A -85,B 0,C 180,E1 -12954.431,E2 -12954.431} C_VEL
LIN {X 0,Y 362.284,Z 655.351,A -85,B 0,C 180,E1 -12957.777,E2 -12957.777} C_VEL
LIN {X 0,Y 362.43,Z 655.334,A -85,B 0,C 180,E1 -12960,E2 -12960} C_VEL
LIN {X 0,Y 362.285,Z 655.355,A -85,B 0,C 180,E1 -12962.224,E2 -12962.224} C_VEL
LIN {X 0,Y 362.174,Z 655.37,A -85,B 0,C 180,E1 -12966.686,E2 -12966.686} C_VEL
LIN {X 0,Y 362.076,Z 655.374,A -85,B 0,C 180,E1 -12968.933,E2 -12968.933} C_VEL
LIN {X 0,Y 361.962,Z 655.393,A -85,B 0,C 180,E1 -12972.332,E2 -12972.332} C_VEL
LIN {X 0,Y 361.964,Z 655.398,A -85,B 0,C 180,E1 -12974.62,E2 -12974.62} C_VEL
LIN {X 0,Y 361.962,Z 655.397,A -85,B 0,C 180,E1 -12978.099,E2 -12978.099} C_VEL
LIN {X 0,Y 361.894,Z 655.404,A -85,B 0,C 180,E1 -12981.653,E2 -12981.653} C_VEL
LIN {X 0,Y 361.93,Z 655.398,A -85,B 0,C 180,E1 -12985.29,E2 -12985.29} C_VEL
LIN {X 0,Y 361.91,Z 655.403,A -85,B 0,C 180,E1 -12987.779,E2 -12987.779} C_VEL
LIN {X 0,Y 361.84,Z 655.413,A -85,B 0,C 180,E1 -12991.629,E2 -12991.629} C_VEL
LIN {X 0,Y 361.876,Z 655.411,A -85,B 0,C 180,E1 -12995.345,E2 -12995.345} C_VEL
LIN {X 0,Y 361.872,Z 655.413,A -85,B 0,C 180,E1 -12999.027,E2 -12999.027} C_VEL
LIN {X 0,Y 361.838,Z 655.409,A -85,B 0,C 180,E1 -13002.829,E2 -13002.829} C_VEL
LIN {X 0,Y 361.861,Z 655.522,A -85,B 0,C 180,E1 -13003.603,E2 -13003.603} C_VEL
LIN {X 0,Y 363.237,Z 661.954,A -85,B 0,C 180,E1 -13006.515,E2 -13006.515} C_VEL
LIN {X 0,Y 364.81,Z 669.854,A -85,B 0,C 180,E1 -13009.777,E2 -13009.777} C_VEL
LIN {X 0,Y 365.821,Z 675.772,A -85,B 0,C 180,E1 -13012.064,E2 -13012.064} C_VEL
LIN {X 0,Y 365.663,Z 679.611,A -85,B 0,C 180,E1 -13013.429,E2 -13013.429} C_VEL
LIN {X 0,Y 364.371,Z 691.14,A -85,B 0,C 180,E1 -13017.312,E2 -13017.312} C_VEL
LIN {X 0,Y 363.302,Z 702.776,A -85,B 0,C 180,E1 -13021.078,E2 -13021.078} C_VEL
LIN {X 0,Y 362.461,Z 714.506,A -85,B 0,C 180,E1 -13024.749,E2 -13024.749} C_VEL
LIN {X 0,Y 361.717,Z 727.91,A -85,B 0,C 180,E1 -13028.847,E2 -13028.847} C_VEL
LIN {X 0,Y 361.6,Z 730.15,A -85,B 0,C 180,E1 -13029.522,E2 -13029.522} C_VEL
LIN {X 0,Y 363.848,Z 745.813,A -85,B 0,C 180,E1 -13030.207,E2 -13030.207} C_VEL
LIN {X 0,Y 365.049,Z 761.893,A -85,B 0,C 180,E1 -13031.089,E2 -13031.089} C_VEL
LIN {X 0,Y 365.763,Z 774.723,A -85,B 0,C 180,E1 -13031.74,E2 -13031.74} C_VEL
LIN {X 0,Y 366.186,Z 782.73,A -85,B 0,C 180,E1 -13032.261,E2 -13032.261} C_VEL
LIN {X 0,Y 365.415,Z 793.573,A -85,B 0,C 180,E1 -13033.088,E2 -13033.088} C_VEL
LIN {X 0,Y 364.387,Z 804.941,A -85,B 0,C 180,E1 -13034.191,E2 -13034.191} C_VEL
LIN {X 0,Y 363.517,Z 815.22,A -85,B 0,C 180,E1 -13035.443,E2 -13035.443} C_VEL
LIN {X 0,Y 362.679,Z 824.448,A -85,B 0,C 180,E1 -13036.838,E2 -13036.838} C_VEL
LIN {X 0,Y 361.767,Z 833.399,A -85,B 0,C 180,E1 -13038.514,E2 -13038.514} C_VEL
LIN {X 0,Y 361.189,Z 840.576,A -85,B 0,C 180,E1 -13040.197,E2 -13040.197} C_VEL
LIN {X 0,Y 360.735,Z 847.074,A -85,B 0,C 180,E1 -13042.161,E2 -13042.161} C_VEL
LIN {X 0,Y 360.53,Z 851.26,A -85,B 0,C 180,E1 -13043.812,E2 -13043.812} C_VEL
LIN {X 0,Y 360.468,Z 854.492,A -85,B 0,C 180,E1 -13045.527,E2 -13045.527} C_VEL
LIN {X 0,Y 360.376,Z 856.049,A -85,B 0,C 180,E1 -13046.645,E2 -13046.645} C_VEL
LIN {X 0,Y 360.384,Z 857.148,A -85,B 0,C 180,E1 -13047.764,E2 -13047.764} C_VEL
LIN {X 0,Y 360.46,Z 857.824,A -85,B 0,C 180,E1 -13048.882,E2 -13048.882} C_VEL
LIN {X 0,Y 360.498,Z 858.102,A -85,B 0,C 180,E1 -13049.999,E2 -13049.999} C_VEL
LIN {X 0,Y 360.443,Z 857.971,A -85,B 0,C 180,E1 -13051.117,E2 -13051.117} C_VEL
LIN {X 0,Y 360.378,Z 857.389,A -85,B 0,C 180,E1 -13052.235,E2 -13052.235} C_VEL
LIN {X 0,Y 360.455,Z 855.024,A -85,B 0,C 180,E1 -13054.472,E2 -13054.472} C_VEL
LIN {X 0,Y 360.492,Z 852.142,A -85,B 0,C 180,E1 -13056.132,E2 -13056.132} C_VEL
LIN {X 0,Y 360.737,Z 848.124,A -85,B 0,C 180,E1 -13057.838,E2 -13057.838} C_VEL
LIN {X 0,Y 361.238,Z 841.984,A -85,B 0,C 180,E1 -13059.801,E2 -13059.801} C_VEL
LIN {X 0,Y 361.838,Z 835.262,A -85,B 0,C 180,E1 -13061.483,E2 -13061.483} C_VEL
LIN {X 0,Y 362.809,Z 826.938,A -85,B 0,C 180,E1 -13063.156,E2 -13063.156} C_VEL
LIN {X 0,Y 363.742,Z 817.249,A -85,B 0,C 180,E1 -13064.712,E2 -13064.712} C_VEL
LIN {X 0,Y 364.852,Z 806.688,A -85,B 0,C 180,E1 -13066.075,E2 -13066.075} C_VEL
LIN {X 0,Y 365.972,Z 796.013,A -85,B 0,C 180,E1 -13067.172,E2 -13067.172} C_VEL
LIN {X 0,Y 366.992,Z 784.352,A -85,B 0,C 180,E1 -13068.117,E2 -13068.117} C_VEL
LIN {X 0,Y 366.568,Z 771.847,A -85,B 0,C 180,E1 -13068.967,E2 -13068.967} C_VEL
LIN {X 0,Y 365.806,Z 758.834,A -85,B 0,C 180,E1 -13069.619,E2 -13069.619} C_VEL
LIN {X 0,Y 364.201,Z 746.099,A -85,B 0,C 180,E1 -13070.102,E2 -13070.102} C_VEL
LIN {X 0,Y 362.715,Z 738.228,A -85,B 0,C 180,E1 -13070.411,E2 -13070.411} C_VEL
LIN {X 0,Y 361.766,Z 729.431,A -85,B 0,C 180,E1 -13071.173,E2 -13071.173} C_VEL
LIN {X 0,Y 362.627,Z 716.232,A -85,B 0,C 180,E1 -13075.237,E2 -13075.237} C_VEL
LIN {X 0,Y 363.601,Z 703.506,A -85,B 0,C 180,E1 -13079.246,E2 -13079.246} C_VEL
LIN {X 0,Y 364.848,Z 690.909,A -85,B 0,C 180,E1 -13083.297,E2 -13083.297} C_VEL
LIN {X 0,Y 365.919,Z 681.096,A -85,B 0,C 180,E1 -13086.54,E2 -13086.54} C_VEL
LIN {X 0,Y 366.036,Z 676.606,A -85,B 0,C 180,E1 -13088.074,E2 -13088.074} C_VEL
LIN {X 0,Y 364.43,Z 668.115,A -85,B 0,C 180,E1 -13091.226,E2 -13091.226} C_VEL
LIN {X 0,Y 362.514,Z 658.598,A -85,B 0,C 180,E1 -13094.958,E2 -13094.958} C_VEL
LIN {X 0,Y 361.911,Z 655.405,A -85,B 0,C 180,E1 -13096.29,E2 -13096.29} C_VEL
LIN {X 0,Y 361.878,Z 655.41,A -85,B 0,C 180,E1 -13100.141,E2 -13100.141} C_VEL
LIN {X 0,Y 361.866,Z 655.406,A -85,B 0,C 180,E1 -13102.982,E2 -13102.982} C_VEL
LIN {X 0,Y 361.855,Z 655.411,A -85,B 0,C 180,E1 -13106.63,E2 -13106.63} C_VEL
LIN {X 0,Y 361.872,Z 655.409,A -85,B 0,C 180,E1 -13109.672,E2 -13109.672} C_VEL
LIN {X 0,Y 361.95,Z 655.398,A -85,B 0,C 180,E1 -13113.475,E2 -13113.475} C_VEL
LIN {X 0,Y 361.885,Z 655.402,A -85,B 0,C 180,E1 -13117.144,E2 -13117.144} C_VEL
LIN {X 0,Y 361.916,Z 655.402,A -85,B 0,C 180,E1 -13120.724,E2 -13120.724} C_VEL
LIN {X 0,Y 361.942,Z 655.4,A -85,B 0,C 180,E1 -13124.226,E2 -13124.226} C_VEL
LIN {X 0,Y 361.995,Z 655.394,A -85,B 0,C 180,E1 -13126.527,E2 -13126.527} C_VEL
LIN {X 0,Y 362.032,Z 655.389,A -85,B 0,C 180,E1 -13129.938,E2 -13129.938} C_VEL
LIN {X 0,Y 362.146,Z 655.378,A -85,B 0,C 180,E1 -13132.192,E2 -13132.192} C_VEL
LIN {X 0,Y 362.113,Z 655.379,A -85,B 0,C 180,E1 -13134.431,E2 -13134.431} C_VEL
LIN {X 0,Y 362.12,Z 655.545,A -85,B 0,C 180,E1 -13136.732,E2 -13136.732} C_VEL
LIN {X 0,Y 363.723,Z 661.523,A -85,B 0,C 180,E1 -13138.893,E2 -13138.893} C_VEL
LIN {X 0,Y 365.058,Z 667.883,A -85,B 0,C 180,E1 -13141.103,E2 -13141.103} C_VEL
LIN {X 0,Y 365.805,Z 672.78,A -85,B 0,C 180,E1 -13142.753,E2 -13142.753} C_VEL
LIN {X 0,Y 365.913,Z 679.666,A -85,B 0,C 180,E1 -13144.958,E2 -13144.958} C_VEL
LIN {X 0,Y 365.402,Z 688.412,A -85,B 0,C 180,E1 -13147.737,E2 -13147.737} C_VEL
LIN {X 0,Y 364.851,Z 699.25,A -85,B 0,C 180,E1 -13151.106,E2 -13151.106} C_VEL
LIN {X 0,Y 364.209,Z 710.168,A -85,B 0,C 180,E1 -13154.528,E2 -13154.528} C_VEL
LIN {X 0,Y 363.573,Z 721.208,A -85,B 0,C 180,E1 -13158.016,E2 -13158.016} C_VEL
LIN {X 0,Y 363.131,Z 729.486,A -85,B 0,C 180,E1 -13160.647,E2 -13160.647} C_VEL
LIN {X 0,Y 366.338,Z 743.115,A -85,B 0,C 180,E1 -13161.34,E2 -13161.34} C_VEL
LIN {X 0,Y 368.427,Z 756.712,A -85,B 0,C 180,E1 -13162.206,E2 -13162.206} C_VEL
LIN {X 0,Y 367.6,Z 768.652,A -85,B 0,C 180,E1 -13163.029,E2 -13163.029} C_VEL
LIN {X 0,Y 366.507,Z 780.043,A -85,B 0,C 180,E1 -13164.047,E2 -13164.047} C_VEL
LIN {X 0,Y 365.341,Z 791.12,A -85,B 0,C 180,E1 -13165.296,E2 -13165.296} C_VEL
LIN {X 0,Y 364.204,Z 800.714,A -85,B 0,C 180,E1 -13166.641,E2 -13166.641} C_VEL
LIN {X 0,Y 363.149,Z 810.194,A -85,B 0,C 180,E1 -13168.304,E2 -13168.304} C_VEL
LIN {X 0,Y 362.2,Z 818.079,A -85,B 0,C 180,E1 -13170.029,E2 -13170.029} C_VEL
LIN {X 0,Y 361.495,Z 825.043,A -85,B 0,C 180,E1 -13171.991,E2 -13171.991} C_VEL
LIN {X 0,Y 360.951,Z 829.859,A -85,B 0,C 180,E1 -13173.744,E2 -13173.744} C_VEL
LIN {X 0,Y 360.515,Z 833.951,A -85,B 0,C 180,E1 -13175.791,E2 -13175.791} C_VEL
LIN {X 0,Y 360.301,Z 835.929,A -85,B 0,C 180,E1 -13177.206,E2 -13177.206} C_VEL
LIN {X 0,Y 360.13,Z 837.258,A -85,B 0,C 180,E1 -13178.685,E2 -13178.685} C_VEL
LIN {X 0,Y 360.049,Z 837.933,A -85,B 0,C 180,E1 -13180.426,E2 -13180.426} C_VEL
LIN {X 0,Y 360.018,Z 837.657,A -85,B 0,C 180,E1 -13182.116,E2 -13182.116} C_VEL
LIN {X 0,Y 360.093,Z 836.496,A -85,B 0,C 180,E1 -13183.77,E2 -13183.77} C_VEL
LIN {X 0,Y 360.287,Z 834.48,A -85,B 0,C 180,E1 -13185.394,E2 -13185.394} C_VEL
LIN {X 0,Y 360.559,Z 831.627,A -85,B 0,C 180,E1 -13186.984,E2 -13186.984} C_VEL
LIN {X 0,Y 360.952,Z 826.606,A -85,B 0,C 180,E1 -13189.001,E2 -13189.001} C_VEL
LIN {X 0,Y 361.422,Z 821.473,A -85,B 0,C 180,E1 -13190.585,E2 -13190.585} C_VEL
LIN {X 0,Y 362.073,Z 815.104,A -85,B 0,C 180,E1 -13192.172,E2 -13192.172} C_VEL
LIN {X 0,Y 362.846,Z 807.328,A -85,B 0,C 180,E1 -13193.747,E2 -13193.747} C_VEL
LIN {X 0,Y 363.784,Z 798.058,A -85,B 0,C 180,E1 -13195.257,E2 -13195.257} C_VEL
LIN {X 0,Y 364.76,Z 788.366,A -85,B 0,C 180,E1 -13196.542,E2 -13196.542} C_VEL
LIN {X 0,Y 365.73,Z 777.314,A -85,B 0,C 180,E1 -13197.728,E2 -13197.728} C_VEL
LIN {X 0,Y 366.76,Z 764.81,A -85,B 0,C 180,E1 -13198.764,E2 -13198.764} C_VEL
LIN {X 0,Y 367.215,Z 755.374,A -85,B 0,C 180,E1 -13199.384,E2 -13199.384} C_VEL
LIN {X 0,Y 365.218,Z 742.373,A -85,B 0,C 180,E1 -13200.148,E2 -13200.148} C_VEL
LIN {X 0,Y 362.632,Z 728.738,A -85,B 0,C 180,E1 -13200.757,E2 -13200.757} C_VEL
LIN {X 0,Y 363.255,Z 717.984,A -85,B 0,C 180,E1 -13204.196,E2 -13204.196} C_VEL
LIN {X 0,Y 363.872,Z 706.126,A -85,B 0,C 180,E1 -13207.986,E2 -13207.986} C_VEL
LIN {X 0,Y 364.428,Z 695.247,A -85,B 0,C 180,E1 -13211.481,E2 -13211.481} C_VEL
LIN {X 0,Y 365.008,Z 684.505,A -85,B 0,C 180,E1 -13214.935,E2 -13214.935} C_VEL
LIN {X 0,Y 365.353,Z 675.694,A -85,B 0,C 180,E1 -13217.785,E2 -13217.785} C_VEL
LIN {X 0,Y 364.683,Z 669.075,A -85,B 0,C 180,E1 -13220.013,E2 -13220.013} C_VEL
LIN {X 0,Y 363,Z 659.513,A -85,B 0,C 180,E1 -13223.33,E2 -13223.33} C_VEL
LIN {X 0,Y 362.046,Z 655.392,A -85,B 0,C 180,E1 -13224.85,E2 -13224.85} C_VEL
LIN {X 0,Y 362.284,Z 655.361,A -85,B 0,C 180,E1 -13227.777,E2 -13227.777} C_VEL
LIN {X 0,Y 362.429,Z 655.342,A -85,B 0,C 180,E1 -13230.001,E2 -13230.001} C_VEL
LIN {X 0,Y 362.284,Z 655.358,A -85,B 0,C 180,E1 -13232.224,E2 -13232.224} C_VEL
LIN {X 0,Y 362.163,Z 655.369,A -85,B 0,C 180,E1 -13236.687,E2 -13236.687} C_VEL
LIN {X 0,Y 362.037,Z 655.385,A -85,B 0,C 180,E1 -13240.062,E2 -13240.062} C_VEL
LIN {X 0,Y 362,Z 655.395,A -85,B 0,C 180,E1 -13243.9,E2 -13243.9} C_VEL
LIN {X 0,Y 361.969,Z 655.401,A -85,B 0,C 180,E1 -13247.939,E2 -13247.939} C_VEL
LIN {X 0,Y 361.947,Z 655.403,A -85,B 0,C 180,E1 -13249.275,E2 -13249.275} C_VEL
LIN {X 0,Y 365.826,Z 668.215,A -85,B 0,C 180,E1 -13250.378,E2 -13250.378} C_VEL
LIN {X 0,Y 367.837,Z 675.756,A -85,B 0,C 180,E1 -13251.139,E2 -13251.139} C_VEL
LIN {X 0,Y 367.09,Z 686.559,A -85,B 0,C 180,E1 -13252.218,E2 -13252.218} C_VEL
LIN {X 0,Y 366.229,Z 697.218,A -85,B 0,C 180,E1 -13253.553,E2 -13253.553} C_VEL
LIN {X 0,Y 365.558,Z 704.756,A -85,B 0,C 180,E1 -13254.698,E2 -13254.698} C_VEL
LIN {X 0,Y 364.526,Z 708.816,A -85,B 0,C 180,E1 -13255.352,E2 -13255.352} C_VEL
LIN {X 0,Y 361.131,Z 715.13,A -85,B 0,C 180,E1 -13256.435,E2 -13256.435} C_VEL
LIN {X 0,Y 357.747,Z 720.858,A -85,B 0,C 180,E1 -13257.609,E2 -13257.609} C_VEL
LIN {X 0,Y 356.752,Z 723.962,A -85,B 0,C 180,E1 -13258.398,E2 -13258.398} C_VEL
LIN {X 0,Y 356.089,Z 729.888,A -85,B 0,C 180,E1 -13260.272,E2 -13260.272} C_VEL
LIN {X 0,Y 355.606,Z 734.569,A -85,B 0,C 180,E1 -13262.25,E2 -13262.25} C_VEL
LIN {X 0,Y 355.272,Z 737.328,A -85,B 0,C 180,E1 -13263.814,E2 -13263.814} C_VEL
LIN {X 0,Y 355.028,Z 739.593,A -85,B 0,C 180,E1 -13265.746,E2 -13265.746} C_VEL
LIN {X 0,Y 354.973,Z 740.748,A -85,B 0,C 180,E1 -13267.862,E2 -13267.862} C_VEL
LIN {X 0,Y 355.091,Z 740.722,A -85,B 0,C 180,E1 -13269.476,E2 -13269.476} C_VEL
LIN {X 0,Y 355.316,Z 739.767,A -85,B 0,C 180,E1 -13271.269,E2 -13271.269} C_VEL
LIN {X 0,Y 355.639,Z 737.883,A -85,B 0,C 180,E1 -13273.015,E2 -13273.015} C_VEL
LIN {X 0,Y 356.327,Z 734.009,A -85,B 0,C 180,E1 -13275.239,E2 -13275.239} C_VEL
LIN {X 0,Y 356.916,Z 730.3,A -85,B 0,C 180,E1 -13276.766,E2 -13276.766} C_VEL
LIN {X 0,Y 357.729,Z 724.443,A -85,B 0,C 180,E1 -13278.658,E2 -13278.658} C_VEL
LIN {X 0,Y 358.612,Z 717.998,A -85,B 0,C 180,E1 -13280.284,E2 -13280.284} C_VEL
LIN {X 0,Y 359.6,Z 710.575,A -85,B 0,C 180,E1 -13281.796,E2 -13281.796} C_VEL
LIN {X 0,Y 360.76,Z 700.961,A -85,B 0,C 180,E1 -13283.378,E2 -13283.378} C_VEL
LIN {X 0,Y 361.791,Z 691.17,A -85,B 0,C 180,E1 -13284.674,E2 -13284.674} C_VEL
LIN {X 0,Y 362.686,Z 680.446,A -85,B 0,C 180,E1 -13285.809,E2 -13285.809} C_VEL
LIN {X 0,Y 360.453,Z 672.065,A -85,B 0,C 180,E1 -13286.745,E2 -13286.745} C_VEL
LIN {X 0,Y 357.025,Z 662.274,A -85,B 0,C 180,E1 -13287.727,E2 -13287.727} C_VEL
LIN {X 0,Y 354.817,Z 656.288,A -85,B 0,C 180,E1 -13288.263,E2 -13288.263} C_VEL
LIN {X 0,Y 354.849,Z 656.285,A -85,B 0,C 180,E1 -13291.619,E2 -13291.619} C_VEL
LIN {X 0,Y 354.9,Z 656.273,A -85,B 0,C 180,E1 -13294.173,E2 -13294.173} C_VEL
LIN {X 0,Y 354.828,Z 656.281,A -85,B 0,C 180,E1 -13297.894,E2 -13297.894} C_VEL
LIN {X 0,Y 354.925,Z 656.278,A -85,B 0,C 180,E1 -13301.891,E2 -13301.891} C_VEL
LIN {X 0,Y 354.944,Z 656.271,A -85,B 0,C 180,E1 -13305.981,E2 -13305.981} C_VEL
LIN {X 0,Y 354.979,Z 656.266,A -85,B 0,C 180,E1 -13309.736,E2 -13309.736} C_VEL
LIN {X 0,Y 355.116,Z 656.243,A -85,B 0,C 180,E1 -13312.037,E2 -13312.037} C_VEL
LIN {X 0,Y 355.094,Z 656.253,A -85,B 0,C 180,E1 -13314.321,E2 -13314.321} C_VEL
LIN {X 0,Y 355.247,Z 656.227,A -85,B 0,C 180,E1 -13317.733,E2 -13317.733} C_VEL
LIN {X 0,Y 355.399,Z 656.21,A -85,B 0,C 180,E1 -13320,E2 -13320} C_VEL
LIN {X 0,Y 355.248,Z 656.232,A -85,B 0,C 180,E1 -13322.268,E2 -13322.268} C_VEL
LIN {X 0,Y 355.14,Z 656.246,A -85,B 0,C 180,E1 -13326.819,E2 -13326.819} C_VEL
LIN {X 0,Y 355.017,Z 656.253,A -85,B 0,C 180,E1 -13329.112,E2 -13329.112} C_VEL
LIN {X 0,Y 354.923,Z 656.268,A -85,B 0,C 180,E1 -13332.581,E2 -13332.581} C_VEL
LIN {X 0,Y 354.891,Z 656.275,A -85,B 0,C 180,E1 -13336.096,E2 -13336.096} C_VEL
LIN {X 0,Y 354.908,Z 656.277,A -85,B 0,C 180,E1 -13338.472,E2 -13338.472} C_VEL
LIN {X 0,Y 354.837,Z 656.286,A -85,B 0,C 180,E1 -13342.106,E2 -13342.106} C_VEL
LIN {X 0,Y 354.901,Z 656.273,A -85,B 0,C 180,E1 -13345.827,E2 -13345.827} C_VEL
LIN {X 0,Y 354.82,Z 656.287,A -85,B 0,C 180,E1 -13349.682,E2 -13349.682} C_VEL
LIN {X 0,Y 354.808,Z 656.29,A -85,B 0,C 180,E1 -13353.702,E2 -13353.702} C_VEL
LIN {X 0,Y 354.8,Z 656.292,A -85,B 0,C 180,E1 -13356.459,E2 -13356.459} C_VEL
LIN {X 0,Y 354.826,Z 656.289,A -85,B 0,C 180,E1 -13359.424,E2 -13359.424} C_VEL
LIN {X 0,Y 354.822,Z 656.345,A -85,B 0,C 180,E1 -13363.049,E2 -13363.049} C_VEL
LIN {X 0,Y 356.534,Z 664.567,A -85,B 0,C 180,E1 -13366.832,E2 -13366.832} C_VEL
LIN {X 0,Y 357.986,Z 672.036,A -85,B 0,C 180,E1 -13369.965,E2 -13369.965} C_VEL
LIN {X 0,Y 358.873,Z 677.495,A -85,B 0,C 180,E1 -13372.124,E2 -13372.124} C_VEL
LIN {X 0,Y 358.436,Z 682.659,A -85,B 0,C 180,E1 -13373.969,E2 -13373.969} C_VEL
LIN {X 0,Y 357.375,Z 692.262,A -85,B 0,C 180,E1 -13377.259,E2 -13377.259} C_VEL
LIN {X 0,Y 356.255,Z 703.871,A -85,B 0,C 180,E1 -13381.097,E2 -13381.097} C_VEL
LIN {X 0,Y 355.386,Z 715.511,A -85,B 0,C 180,E1 -13384.838,E2 -13384.838} C_VEL
LIN {X 0,Y 354.597,Z 729.176,A -85,B 0,C 180,E1 -13389.058,E2 -13389.058} C_VEL
LIN {X 0,Y 356.84,Z 744.154,A -85,B 0,C 180,E1 -13389.726,E2 -13389.726} C_VEL
LIN {X 0,Y 357.962,Z 757.334,A -85,B 0,C 180,E1 -13390.502,E2 -13390.502} C_VEL
LIN {X 0,Y 358.27,Z 763.263,A -85,B 0,C 180,E1 -13390.831,E2 -13390.831} C_VEL
LIN {X 0,Y 358.92,Z 776.029,A -85,B 0,C 180,E1 -13391.515,E2 -13391.515} C_VEL
LIN {X 0,Y 359.25,Z 783.845,A -85,B 0,C 180,E1 -13392.054,E2 -13392.054} C_VEL
LIN {X 0,Y 358.308,Z 795.974,A -85,B 0,C 180,E1 -13393.036,E2 -13393.036} C_VEL
LIN {X 0,Y 357.319,Z 806.867,A -85,B 0,C 180,E1 -13394.165,E2 -13394.165} C_VEL
LIN {X 0,Y 356.428,Z 816.674,A -85,B 0,C 180,E1 -13395.439,E2 -13395.439} C_VEL
LIN {X 0,Y 355.567,Z 825.616,A -85,B 0,C 180,E1 -13396.861,E2 -13396.861} C_VEL
LIN {X 0,Y 354.615,Z 834.318,A -85,B 0,C 180,E1 -13398.569,E2 -13398.569} C_VEL
LIN {X 0,Y 354.062,Z 841.235,A -85,B 0,C 180,E1 -13400.286,E2 -13400.286} C_VEL
LIN {X 0,Y 353.688,Z 846.75,A -85,B 0,C 180,E1 -13402.004,E2 -13402.004} C_VEL
LIN {X 0,Y 353.457,Z 851.25,A -85,B 0,C 180,E1 -13403.818,E2 -13403.818} C_VEL
LIN {X 0,Y 353.377,Z 854.225,A -85,B 0,C 180,E1 -13405.437,E2 -13405.437} C_VEL
LIN {X 0,Y 353.297,Z 855.795,A -85,B 0,C 180,E1 -13406.578,E2 -13406.578} C_VEL
LIN {X 0,Y 353.285,Z 856.918,A -85,B 0,C 180,E1 -13407.719,E2 -13407.719} C_VEL
LIN {X 0,Y 353.359,Z 857.605,A -85,B 0,C 180,E1 -13408.86,E2 -13408.86} C_VEL
LIN {X 0,Y 353.401,Z 857.895,A -85,B 0,C 180,E1 -13409.999,E2 -13409.999} C_VEL
LIN {X 0,Y 353.342,Z 857.781,A -85,B 0,C 180,E1 -13411.139,E2 -13411.139} C_VEL
LIN {X 0,Y 353.28,Z 857.217,A -85,B 0,C 180,E1 -13412.28,E2 -13412.28} C_VEL
LIN {X 0,Y 353.291,Z 856.246,A -85,B 0,C 180,E1 -13413.421,E2 -13413.421} C_VEL
LIN {X 0,Y 353.365,Z 854.873,A -85,B 0,C 180,E1 -13414.562,E2 -13414.562} C_VEL
LIN {X 0,Y 353.39,Z 852.346,A -85,B 0,C 180,E1 -13416.081,E2 -13416.081} C_VEL
LIN {X 0,Y 353.694,Z 848.017,A -85,B 0,C 180,E1 -13417.995,E2 -13417.995} C_VEL
LIN {X 0,Y 354.217,Z 841.916,A -85,B 0,C 180,E1 -13419.997,E2 -13419.997} C_VEL
LIN {X 0,Y 354.861,Z 835.221,A -85,B 0,C 180,E1 -13421.712,E2 -13421.712} C_VEL
LIN {X 0,Y 355.871,Z 826.955,A -85,B 0,C 180,E1 -13423.417,E2 -13423.417} C_VEL
LIN {X 0,Y 356.737,Z 818.483,A -85,B 0,C 180,E1 -13424.839,E2 -13424.839} C_VEL
LIN {X 0,Y 357.905,Z 808.052,A -85,B 0,C 180,E1 -13426.249,E2 -13426.249} C_VEL
LIN {X 0,Y 359.22,Z 796.359,A -85,B 0,C 180,E1 -13427.505,E2 -13427.505} C_VEL
LIN {X 0,Y 360.268,Z 784.764,A -85,B 0,C 180,E1 -13428.474,E2 -13428.474} C_VEL
LIN {X 0,Y 359.865,Z 771.668,A -85,B 0,C 180,E1 -13429.39,E2 -13429.39} C_VEL
LIN {X 0,Y 359.124,Z 758.687,A -85,B 0,C 180,E1 -13430.056,E2 -13430.056} C_VEL
LIN {X 0,Y 357.582,Z 746.68,A -85,B 0,C 180,E1 -13430.538,E2 -13430.538} C_VEL
LIN {X 0,Y 355.954,Z 737.94,A -85,B 0,C 180,E1 -13430.906,E2 -13430.906} C_VEL
LIN {X 0,Y 354.808,Z 727.431,A -85,B 0,C 180,E1 -13431.89,E2 -13431.89} C_VEL
LIN {X 0,Y 355.648,Z 715.185,A -85,B 0,C 180,E1 -13435.768,E2 -13435.768} C_VEL
LIN {X 0,Y 356.616,Z 703.558,A -85,B 0,C 180,E1 -13439.516,E2 -13439.516} C_VEL
LIN {X 0,Y 357.837,Z 691.87,A -85,B 0,C 180,E1 -13443.361,E2 -13443.361} C_VEL
LIN {X 0,Y 359.017,Z 681.344,A -85,B 0,C 180,E1 -13446.916,E2 -13446.916} C_VEL
LIN {X 0,Y 358.912,Z 677.042,A -85,B 0,C 180,E1 -13448.44,E2 -13448.44} C_VEL
LIN {X 0,Y 357.162,Z 667.707,A -85,B 0,C 180,E1 -13451.991,E2 -13451.991} C_VEL
LIN {X 0,Y 355.087,Z 657.471,A -85,B 0,C 180,E1 -13456.153,E2 -13456.153} C_VEL
LIN {X 0,Y 354.878,Z 656.283,A -85,B 0,C 180,E1 -13456.673,E2 -13456.673} C_VEL
LIN {X 0,Y 354.853,Z 656.283,A -85,B 0,C 180,E1 -13459.188,E2 -13459.188} C_VEL
LIN {X 0,Y 354.806,Z 656.283,A -85,B 0,C 180,E1 -13462.401,E2 -13462.401} C_VEL
LIN {X 0,Y 354.808,Z 656.283,A -85,B 0,C 180,E1 -13464.94,E2 -13464.94} C_VEL
LIN {X 0,Y 354.789,Z 656.284,A -85,B 0,C 180,E1 -13468.404,E2 -13468.404} C_VEL
LIN {X 0,Y 354.85,Z 656.278,A -85,B 0,C 180,E1 -13471.619,E2 -13471.619} C_VEL
LIN {X 0,Y 354.895,Z 656.272,A -85,B 0,C 180,E1 -13474.172,E2 -13474.172} C_VEL
LIN {X 0,Y 354.83,Z 656.284,A -85,B 0,C 180,E1 -13477.893,E2 -13477.893} C_VEL
LIN {X 0,Y 354.918,Z 656.272,A -85,B 0,C 180,E1 -13481.891,E2 -13481.891} C_VEL
LIN {X 0,Y 354.938,Z 656.273,A -85,B 0,C 180,E1 -13485.98,E2 -13485.98} C_VEL
LIN {X 0,Y 354.978,Z 656.267,A -85,B 0,C 180,E1 -13489.736,E2 -13489.736} C_VEL
LIN {X 0,Y 355.109,Z 656.254,A -85,B 0,C 180,E1 -13492.037,E2 -13492.037} C_VEL
LIN {X 0,Y 355.087,Z 656.255,A -85,B 0,C 180,E1 -13494.32,E2 -13494.32} C_VEL
LIN {X 0,Y 354.972,Z 656.424,A -85,B 0,C 180,E1 -13495.955,E2 -13495.955} C_VEL
LIN {X 0,Y 356.822,Z 662.668,A -85,B 0,C 180,E1 -13498.307,E2 -13498.307} C_VEL
LIN {X 0,Y 358.19,Z 668.947,A -85,B 0,C 180,E1 -13500.562,E2 -13500.562} C_VEL
LIN {X 0,Y 359.114,Z 675.44,A -85,B 0,C 180,E1 -13502.804,E2 -13502.804} C_VEL
LIN {X 0,Y 359.119,Z 682.309,A -85,B 0,C 180,E1 -13505.052,E2 -13505.052} C_VEL
LIN {X 0,Y 358.424,Z 692.994,A -85,B 0,C 180,E1 -13508.456,E2 -13508.456} C_VEL
LIN {X 0,Y 357.828,Z 703.874,A -85,B 0,C 180,E1 -13511.901,E2 -13511.901} C_VEL
LIN {X 0,Y 357.125,Z 714.713,A -85,B 0,C 180,E1 -13515.362,E2 -13515.362} C_VEL
LIN {X 0,Y 356.483,Z 726.435,A -85,B 0,C 180,E1 -13519.133,E2 -13519.133} C_VEL
LIN {X 0,Y 356.282,Z 729.625,A -85,B 0,C 180,E1 -13520.156,E2 -13520.156} C_VEL
LIN {X 0,Y 359.67,Z 743.865,A -85,B 0,C 180,E1 -13520.929,E2 -13520.929} C_VEL
LIN {X 0,Y 361.712,Z 757.273,A -85,B 0,C 180,E1 -13521.814,E2 -13521.814} C_VEL
LIN {X 0,Y 360.966,Z 768.597,A -85,B 0,C 180,E1 -13522.615,E2 -13522.615} C_VEL
LIN {X 0,Y 359.822,Z 780.192,A -85,B 0,C 180,E1 -13523.665,E2 -13523.665} C_VEL
LIN {X 0,Y 358.604,Z 791.161,A -85,B 0,C 180,E1 -13524.92,E2 -13524.92} C_VEL
LIN {X 0,Y 357.448,Z 800.583,A -85,B 0,C 180,E1 -13526.256,E2 -13526.256} C_VEL
LIN {X 0,Y 356.386,Z 809.528,A -85,B 0,C 180,E1 -13527.835,E2 -13527.835} C_VEL
LIN {X 0,Y 355.349,Z 817.737,A -85,B 0,C 180,E1 -13529.633,E2 -13529.633} C_VEL
LIN {X 0,Y 354.577,Z 824.534,A -85,B 0,C 180,E1 -13531.54,E2 -13531.54} C_VEL
LIN {X 0,Y 353.922,Z 829.897,A -85,B 0,C 180,E1 -13533.489,E2 -13533.489} C_VEL
LIN {X 0,Y 353.484,Z 833.769,A -85,B 0,C 180,E1 -13535.398,E2 -13535.398} C_VEL
LIN {X 0,Y 353.196,Z 836.327,A -85,B 0,C 180,E1 -13537.258,E2 -13537.258} C_VEL
LIN {X 0,Y 353.004,Z 837.755,A -85,B 0,C 180,E1 -13539.064,E2 -13539.064} C_VEL
LIN {X 0,Y 352.933,Z 838.136,A -85,B 0,C 180,E1 -13541.081,E2 -13541.081} C_VEL
LIN {X 0,Y 352.948,Z 837.618,A -85,B 0,C 180,E1 -13542.611,E2 -13542.611} C_VEL
LIN {X 0,Y 353.117,Z 835.355,A -85,B 0,C 180,E1 -13544.954,E2 -13544.954} C_VEL
LIN {X 0,Y 353.373,Z 832.761,A -85,B 0,C 180,E1 -13546.569,E2 -13546.569} C_VEL
LIN {X 0,Y 353.691,Z 829.048,A -85,B 0,C 180,E1 -13548.269,E2 -13548.269} C_VEL
LIN {X 0,Y 354.208,Z 823.432,A -85,B 0,C 180,E1 -13550.218,E2 -13550.218} C_VEL
LIN {X 0,Y 354.814,Z 817.716,A -85,B 0,C 180,E1 -13551.774,E2 -13551.774} C_VEL
LIN {X 0,Y 355.491,Z 810.768,A -85,B 0,C 180,E1 -13553.321,E2 -13553.321} C_VEL
LIN {X 0,Y 356.471,Z 801.662,A -85,B 0,C 180,E1 -13554.957,E2 -13554.957} C_VEL
LIN {X 0,Y 357.534,Z 791.662,A -85,B 0,C 180,E1 -13556.41,E2 -13556.41} C_VEL
LIN {X 0,Y 358.577,Z 780.752,A -85,B 0,C 180,E1 -13557.674,E2 -13557.674} C_VEL
LIN {X 0,Y 359.552,Z 769.409,A -85,B 0,C 180,E1 -13558.72,E2 -13558.72} C_VEL
LIN {X 0,Y 360.434,Z 758.003,A -85,B 0,C 180,E1 -13559.539,E2 -13559.539} C_VEL
LIN {X 0,Y 358.835,Z 746.043,A -85,B 0,C 180,E1 -13560.291,E2 -13560.291} C_VEL
LIN {X 0,Y 356.325,Z 732.424,A -85,B 0,C 180,E1 -13560.943,E2 -13560.943} C_VEL
LIN {X 0,Y 355.635,Z 728.949,A -85,B 0,C 180,E1 -13561.084,E2 -13561.084} C_VEL
LIN {X 0,Y 356.265,Z 719.067,A -85,B 0,C 180,E1 -13564.28,E2 -13564.28} C_VEL
LIN {X 0,Y 356.898,Z 707.492,A -85,B 0,C 180,E1 -13568.029,E2 -13568.029} C_VEL
LIN {X 0,Y 357.511,Z 696.269,A -85,B 0,C 180,E1 -13571.668,E2 -13571.668} C_VEL
LIN {X 0,Y 358.119,Z 685.351,A -85,B 0,C 180,E1 -13575.22,E2 -13575.22} C_VEL
LIN {X 0,Y 358.419,Z 676.52,A -85,B 0,C 180,E1 -13578.119,E2 -13578.119} C_VEL
LIN {X 0,Y 357.672,Z 669.895,A -85,B 0,C 180,E1 -13580.386,E2 -13580.386} C_VEL
LIN {X 0,Y 355.953,Z 660.293,A -85,B 0,C 180,E1 -13583.766,E2 -13583.766} C_VEL
LIN {X 0,Y 354.958,Z 656.278,A -85,B 0,C 180,E1 -13585.245,E2 -13585.245} C_VEL
LIN {X 0,Y 355.247,Z 656.237,A -85,B 0,C 180,E1 -13587.733,E2 -13587.733} C_VEL
LIN {X 0,Y 355.399,Z 656.217,A -85,B 0,C 180,E1 -13590.001,E2 -13590.001} C_VEL
LIN {X 0,Y 355.247,Z 656.235,A -85,B 0,C 180,E1 -13592.268,E2 -13592.268} C_VEL
LIN {X 0,Y 355.127,Z 656.245,A -85,B 0,C 180,E1 -13596.82,E2 -13596.82} C_VEL
LIN {X 0,Y 354.984,Z 656.264,A -85,B 0,C 180,E1 -13600.264,E2 -13600.264} C_VEL
LIN {X 0,Y 354.945,Z 656.273,A -85,B 0,C 180,E1 -13604.02,E2 -13604.02} C_VEL
LIN {X 0,Y 354.925,Z 656.277,A -85,B 0,C 180,E1 -13608.109,E2 -13608.109} C_VEL
LIN {X 0,Y 354.925,Z 656.441,A -85,B 0,C 180,E1 -13608.958,E2 -13608.958} C_VEL
LIN {X 0,Y 358.409,Z 667.689,A -85,B 0,C 180,E1 -13609.92,E2 -13609.92} C_VEL
LIN {X 0,Y 360.883,Z 676.501,A -85,B 0,C 180,E1 -13610.819,E2 -13610.819} C_VEL
LIN {X 0,Y 360.761,Z 681.177,A -85,B 0,C 180,E1 -13611.275,E2 -13611.275} C_VEL
LIN {X 0,Y 359.9,Z 692.435,A -85,B 0,C 180,E1 -13612.534,E2 -13612.534} C_VEL
LIN {X 0,Y 358.955,Z 702.752,A -85,B 0,C 180,E1 -13613.99,E2 -13613.99} C_VEL
LIN {X 0,Y 358.077,Z 711.864,A -85,B 0,C 180,E1 -13615.582,E2 -13615.582} C_VEL
LIN {X 0,Y 357.177,Z 719.672,A -85,B 0,C 180,E1 -13617.272,E2 -13617.272} C_VEL
LIN {X 0,Y 356.752,Z 723.962,A -85,B 0,C 180,E1 -13618.398,E2 -13618.398} C_VEL
LIN {X 0,Y 355.778,Z 726.871,A -85,B 0,C 180,E1 -13619.212,E2 -13619.212} C_VEL
LIN {X 0,Y 352.503,Z 731.268,A -85,B 0,C 180,E1 -13620.551,E2 -13620.551} C_VEL
LIN {X 0,Y 349.292,Z 735.057,A -85,B 0,C 180,E1 -13621.959,E2 -13621.959} C_VEL
LIN {X 0,Y 348.435,Z 736.868,A -85,B 0,C 180,E1 -13622.869,E2 -13622.869} C_VEL
LIN {X 0,Y 348.172,Z 739.204,A -85,B 0,C 180,E1 -13624.416,E2 -13624.416} C_VEL
LIN {X 0,Y 347.981,Z 740.906,A -85,B 0,C 180,E1 -13626.113,E2 -13626.113} C_VEL
LIN {X 0,Y 347.953,Z 741.809,A -85,B 0,C 180,E1 -13628.027,E2 -13628.027} C_VEL
LIN {X 0,Y 348.171,Z 741.533,A -85,B 0,C 180,E1 -13630.236,E2 -13630.236} C_VEL
LIN {X 0,Y 348.385,Z 740.502,A -85,B 0,C 180,E1 -13631.737,E2 -13631.737} C_VEL
LIN {X 0,Y 348.955,Z 737.546,A -85,B 0,C 180,E1 -13634.084,E2 -13634.084} C_VEL
LIN {X 0,Y 349.508,Z 734.409,A -85,B 0,C 180,E1 -13635.73,E2 -13635.73} C_VEL
LIN {X 0,Y 350.167,Z 730.324,A -85,B 0,C 180,E1 -13637.368,E2 -13637.368} C_VEL
LIN {X 0,Y 350.952,Z 725.221,A -85,B 0,C 180,E1 -13638.987,E2 -13638.987} C_VEL
LIN {X 0,Y 352.031,Z 717.754,A -85,B 0,C 180,E1 -13640.853,E2 -13640.853} C_VEL
LIN {X 0,Y 353.235,Z 708.88,A -85,B 0,C 180,E1 -13642.611,E2 -13642.611} C_VEL
LIN {X 0,Y 354.295,Z 700.365,A -85,B 0,C 180,E1 -13643.964,E2 -13643.964} C_VEL
LIN {X 0,Y 355.417,Z 689.535,A -85,B 0,C 180,E1 -13645.355,E2 -13645.355} C_VEL
LIN {X 0,Y 355.967,Z 681.33,A -85,B 0,C 180,E1 -13646.228,E2 -13646.228} C_VEL
LIN {X 0,Y 352.738,Z 670.576,A -85,B 0,C 180,E1 -13647.456,E2 -13647.456} C_VEL
LIN {X 0,Y 348.565,Z 659.639,A -85,B 0,C 180,E1 -13648.553,E2 -13648.553} C_VEL
LIN {X 0,Y 347.77,Z 657.167,A -85,B 0,C 180,E1 -13648.77,E2 -13648.77} C_VEL
LIN {X 0,Y 347.852,Z 657.156,A -85,B 0,C 180,E1 -13652.745,E2 -13652.745} C_VEL
LIN {X 0,Y 347.787,Z 657.158,A -85,B 0,C 180,E1 -13656.162,E2 -13656.162} C_VEL
LIN {X 0,Y 347.814,Z 657.162,A -85,B 0,C 180,E1 -13659.91,E2 -13659.91} C_VEL
LIN {X 0,Y 347.869,Z 657.153,A -85,B 0,C 180,E1 -13662.36,E2 -13662.36} C_VEL
LIN {X 0,Y 347.899,Z 657.149,A -85,B 0,C 180,E1 -13665.971,E2 -13665.971} C_VEL
LIN {X 0,Y 347.93,Z 657.142,A -85,B 0,C 180,E1 -13669.526,E2 -13669.526} C_VEL
LIN {X 0,Y 348.076,Z 657.121,A -85,B 0,C 180,E1 -13671.875,E2 -13671.875} C_VEL
LIN {X 0,Y 348.069,Z 657.13,A -85,B 0,C 180,E1 -13674.206,E2 -13674.206} C_VEL
LIN {X 0,Y 348.21,Z 657.103,A -85,B 0,C 180,E1 -13677.687,E2 -13677.687} C_VEL
LIN {X 0,Y 348.348,Z 657.088,A -85,B 0,C 180,E1 -13680,E2 -13680} C_VEL
LIN {X 0,Y 348.21,Z 657.109,A -85,B 0,C 180,E1 -13682.314,E2 -13682.314} C_VEL
LIN {X 0,Y 348.108,Z 657.121,A -85,B 0,C 180,E1 -13686.958,E2 -13686.958} C_VEL
LIN {X 0,Y 347.969,Z 657.131,A -85,B 0,C 180,E1 -13689.299,E2 -13689.299} C_VEL
LIN {X 0,Y 347.892,Z 657.142,A -85,B 0,C 180,E1 -13692.84,E2 -13692.84} C_VEL
LIN {X 0,Y 347.841,Z 657.151,A -85,B 0,C 180,E1 -13696.431,E2 -13696.431} C_VEL
LIN {X 0,Y 347.858,Z 657.151,A -85,B 0,C 180,E1 -13698.86,E2 -13698.86} C_VEL
LIN {X 0,Y 347.776,Z 657.161,A -85,B 0,C 180,E1 -13702.579,E2 -13702.579} C_VEL
LIN {X 0,Y 347.814,Z 657.157,A -85,B 0,C 180,E1 -13705.108,E2 -13705.108} C_VEL
LIN {X 0,Y 347.81,Z 657.16,A -85,B 0,C 180,E1 -13707.694,E2 -13707.694} C_VEL
LIN {X 0,Y 347.751,Z 657.167,A -85,B 0,C 180,E1 -13710.348,E2 -13710.348} C_VEL
LIN {X 0,Y 347.75,Z 657.171,A -85,B 0,C 180,E1 -13714.044,E2 -13714.044} C_VEL
LIN {X 0,Y 347.764,Z 657.17,A -85,B 0,C 180,E1 -13717.321,E2 -13717.321} C_VEL
LIN {X 0,Y 347.735,Z 657.173,A -85,B 0,C 180,E1 -13720.297,E2 -13720.297} C_VEL
LIN {X 0,Y 347.777,Z 657.292,A -85,B 0,C 180,E1 -13722.51,E2 -13722.51} C_VEL
LIN {X 0,Y 349.174,Z 663.898,A -85,B 0,C 180,E1 -13725.689,E2 -13725.689} C_VEL
LIN {X 0,Y 350.657,Z 671.361,A -85,B 0,C 180,E1 -13728.976,E2 -13728.976} C_VEL
LIN {X 0,Y 351.832,Z 678.105,A -85,B 0,C 180,E1 -13731.739,E2 -13731.739} C_VEL
LIN {X 0,Y 351.797,Z 681.55,A -85,B 0,C 180,E1 -13733.044,E2 -13733.044} C_VEL
LIN {X 0,Y 350.57,Z 691.441,A -85,B 0,C 180,E1 -13736.543,E2 -13736.543} C_VEL
LIN {X 0,Y 349.361,Z 702.98,A -85,B 0,C 180,E1 -13740.471,E2 -13740.471} C_VEL
LIN {X 0,Y 348.552,Z 712.672,A -85,B 0,C 180,E1 -13743.666,E2 -13743.666} C_VEL
LIN {X 0,Y 347.859,Z 722.352,A -85,B 0,C 180,E1 -13746.798,E2 -13746.798} C_VEL
LIN {X 0,Y 347.574,Z 727.893,A -85,B 0,C 180,E1 -13748.55,E2 -13748.55} C_VEL
LIN {X 0,Y 349.824,Z 742.505,A -85,B 0,C 180,E1 -13749.224,E2 -13749.224} C_VEL
LIN {X 0,Y 350.926,Z 754.607,A -85,B 0,C 180,E1 -13749.942,E2 -13749.942} C_VEL
LIN {X 0,Y 351.4,Z 762.721,A -85,B 0,C 180,E1 -13750.475,E2 -13750.475} C_VEL
LIN {X 0,Y 351.996,Z 775.273,A -85,B 0,C 180,E1 -13751.155,E2 -13751.155} C_VEL
LIN {X 0,Y 352.325,Z 784.949,A -85,B 0,C 180,E1 -13751.839,E2 -13751.839} C_VEL
LIN {X 0,Y 351.349,Z 796.809,A -85,B 0,C 180,E1 -13752.839,E2 -13752.839} C_VEL
LIN {X 0,Y 350.306,Z 807.659,A -85,B 0,C 180,E1 -13754.016,E2 -13754.016} C_VEL
LIN {X 0,Y 349.322,Z 818.094,A -85,B 0,C 180,E1 -13755.434,E2 -13755.434} C_VEL
LIN {X 0,Y 348.438,Z 826.769,A -85,B 0,C 180,E1 -13756.884,E2 -13756.884} C_VEL
LIN {X 0,Y 347.494,Z 835.15,A -85,B 0,C 180,E1 -13758.627,E2 -13758.627} C_VEL
LIN {X 0,Y 346.926,Z 841.88,A -85,B 0,C 180,E1 -13760.379,E2 -13760.379} C_VEL
LIN {X 0,Y 346.539,Z 848.005,A -85,B 0,C 180,E1 -13762.424,E2 -13762.424} C_VEL
LIN {X 0,Y 346.339,Z 851.942,A -85,B 0,C 180,E1 -13764.176,E2 -13764.176} C_VEL
LIN {X 0,Y 346.291,Z 853.953,A -85,B 0,C 180,E1 -13765.343,E2 -13765.343} C_VEL
LIN {X 0,Y 346.219,Z 855.537,A -85,B 0,C 180,E1 -13766.508,E2 -13766.508} C_VEL
LIN {X 0,Y 346.191,Z 856.686,A -85,B 0,C 180,E1 -13767.672,E2 -13767.672} C_VEL
LIN {X 0,Y 346.258,Z 857.386,A -85,B 0,C 180,E1 -13768.836,E2 -13768.836} C_VEL
LIN {X 0,Y 346.303,Z 857.687,A -85,B 0,C 180,E1 -13769.999,E2 -13769.999} C_VEL
LIN {X 0,Y 346.241,Z 857.587,A -85,B 0,C 180,E1 -13771.162,E2 -13771.162} C_VEL
LIN {X 0,Y 346.185,Z 857.045,A -85,B 0,C 180,E1 -13772.326,E2 -13772.326} C_VEL
LIN {X 0,Y 346.213,Z 856.085,A -85,B 0,C 180,E1 -13773.491,E2 -13773.491} C_VEL
LIN {X 0,Y 346.278,Z 854.722,A -85,B 0,C 180,E1 -13774.656,E2 -13774.656} C_VEL
LIN {X 0,Y 346.307,Z 852.495,A -85,B 0,C 180,E1 -13776.056,E2 -13776.056} C_VEL
LIN {X 0,Y 346.644,Z 847.919,A -85,B 0,C 180,E1 -13778.158,E2 -13778.158} C_VEL
LIN {X 0,Y 347.09,Z 842.847,A -85,B 0,C 180,E1 -13779.91,E2 -13779.91} C_VEL
LIN {X 0,Y 347.725,Z 836.469,A -85,B 0,C 180,E1 -13781.66,E2 -13781.66} C_VEL
LIN {X 0,Y 348.752,Z 828.496,A -85,B 0,C 180,E1 -13783.399,E2 -13783.399} C_VEL
LIN {X 0,Y 349.684,Z 820.391,A -85,B 0,C 180,E1 -13784.847,E2 -13784.847} C_VEL
LIN {X 0,Y 350.88,Z 810.536,A -85,B 0,C 180,E1 -13786.284,E2 -13786.284} C_VEL
LIN {X 0,Y 352.136,Z 799.471,A -85,B 0,C 180,E1 -13787.569,E2 -13787.569} C_VEL
LIN {X 0,Y 353.425,Z 787.03,A -85,B 0,C 180,E1 -13788.701,E2 -13788.701} C_VEL
LIN {X 0,Y 353.322,Z 776.128,A -85,B 0,C 180,E1 -13789.534,E2 -13789.534} C_VEL
LIN {X 0,Y 352.829,Z 763.101,A -85,B 0,C 180,E1 -13790.3,E2 -13790.3} C_VEL
LIN {X 0,Y 351.674,Z 751.542,A -85,B 0,C 180,E1 -13790.825,E2 -13790.825} C_VEL
LIN {X 0,Y 349.257,Z 738.29,A -85,B 0,C 180,E1 -13791.371,E2 -13791.371} C_VEL
LIN {X 0,Y 347.866,Z 725.441,A -85,B 0,C 180,E1 -13792.651,E2 -13792.651} C_VEL
LIN {X 0,Y 348.683,Z 714.113,A -85,B 0,C 180,E1 -13796.322,E2 -13796.322} C_VEL
LIN {X 0,Y 349.745,Z 702.313,A -85,B 0,C 180,E1 -13800.223,E2 -13800.223} C_VEL
LIN {X 0,Y 350.814,Z 692.796,A -85,B 0,C 180,E1 -13803.429,E2 -13803.429} C_VEL
LIN {X 0,Y 352.016,Z 682.441,A -85,B 0,C 180,E1 -13807.003,E2 -13807.003} C_VEL
LIN {X 0,Y 352.041,Z 679.036,A -85,B 0,C 180,E1 -13808.233,E2 -13808.233} C_VEL
LIN {X 0,Y 350.486,Z 670.73,A -85,B 0,C 180,E1 -13811.43,E2 -13811.43} C_VEL
LIN {X 0,Y 348.69,Z 661.643,A -85,B 0,C 180,E1 -13815.134,E2 -13815.134} C_VEL
LIN {X 0,Y 347.799,Z 657.163,A -85,B 0,C 180,E1 -13817.099,E2 -13817.099} C_VEL
LIN {X 0,Y 347.783,Z 657.166,A -85,B 0,C 180,E1 -13820.165,E2 -13820.165} C_VEL
LIN {X 0,Y 347.786,Z 657.165,A -85,B 0,C 180,E1 -13824.124,E2 -13824.124} C_VEL
LIN {X 0,Y 347.735,Z 657.164,A -85,B 0,C 180,E1 -13828.085,E2 -13828.085} C_VEL
LIN {X 0,Y 347.802,Z 657.156,A -85,B 0,C 180,E1 -13830.99,E2 -13830.99} C_VEL
LIN {X 0,Y 347.828,Z 657.155,A -85,B 0,C 180,E1 -13833.607,E2 -13833.607} C_VEL
LIN {X 0,Y 347.784,Z 657.163,A -85,B 0,C 180,E1 -13836.161,E2 -13836.161} C_VEL
LIN {X 0,Y 347.812,Z 657.155,A -85,B 0,C 180,E1 -13839.909,E2 -13839.909} C_VEL
LIN {X 0,Y 347.862,Z 657.149,A -85,B 0,C 180,E1 -13842.359,E2 -13842.359} C_VEL
LIN {X 0,Y 347.892,Z 657.151,A -85,B 0,C 180,E1 -13845.97,E2 -13845.97} C_VEL
LIN {X 0,Y 347.929,Z 657.144,A -85,B 0,C 180,E1 -13849.525,E2 -13849.525} C_VEL
LIN {X 0,Y 348.069,Z 657.13,A -85,B 0,C 180,E1 -13851.874,E2 -13851.874} C_VEL
LIN {X 0,Y 347.953,Z 657.143,A -85,B 0,C 180,E1 -13854.785,E2 -13854.785} C_VEL
LIN {X 0,Y 347.928,Z 657.167,A -85,B 0,C 180,E1 -13855.075,E2 -13855.075} C_VEL
LIN {X 0,Y 350.288,Z 665.406,A -85,B 0,C 180,E1 -13858.275,E2 -13858.275} C_VEL
LIN {X 0,Y 351.582,Z 671.511,A -85,B 0,C 180,E1 -13860.515,E2 -13860.515} C_VEL
LIN {X 0,Y 352.445,Z 678.186,A -85,B 0,C 180,E1 -13862.857,E2 -13862.857} C_VEL
LIN {X 0,Y 352.323,Z 685.07,A -85,B 0,C 180,E1 -13865.15,E2 -13865.15} C_VEL
LIN {X 0,Y 351.582,Z 695.87,A -85,B 0,C 180,E1 -13868.622,E2 -13868.622} C_VEL
LIN {X 0,Y 350.931,Z 706.719,A -85,B 0,C 180,E1 -13872.139,E2 -13872.139} C_VEL
LIN {X 0,Y 350.154,Z 718.062,A -85,B 0,C 180,E1 -13875.821,E2 -13875.821} C_VEL
LIN {X 0,Y 349.485,Z 730.105,A -85,B 0,C 180,E1 -13879.684,E2 -13879.684} C_VEL
LIN {X 0,Y 352.663,Z 743.201,A -85,B 0,C 180,E1 -13880.396,E2 -13880.396} C_VEL
LIN {X 0,Y 354.675,Z 755.192,A -85,B 0,C 180,E1 -13881.2,E2 -13881.2} C_VEL
LIN {X 0,Y 355.121,Z 759.83,A -85,B 0,C 180,E1 -13881.545,E2 -13881.545} C_VEL
LIN {X 0,Y 354.038,Z 771.902,A -85,B 0,C 180,E1 -13882.466,E2 -13882.466} C_VEL
LIN {X 0,Y 352.795,Z 783.504,A -85,B 0,C 180,E1 -13883.603,E2 -13883.603} C_VEL
LIN {X 0,Y 351.503,Z 794.369,A -85,B 0,C 180,E1 -13884.959,E2 -13884.959} C_VEL
LIN {X 0,Y 350.312,Z 803.419,A -85,B 0,C 180,E1 -13886.351,E2 -13886.351} C_VEL
LIN {X 0,Y 349.216,Z 811.908,A -85,B 0,C 180,E1 -13887.958,E2 -13887.958} C_VEL
LIN {X 0,Y 348.186,Z 819.59,A -85,B 0,C 180,E1 -13889.782,E2 -13889.782} C_VEL
LIN {X 0,Y 347.385,Z 826.337,A -85,B 0,C 180,E1 -13891.822,E2 -13891.822} C_VEL
LIN {X 0,Y 346.764,Z 831.252,A -85,B 0,C 180,E1 -13893.804,E2 -13893.804} C_VEL
LIN {X 0,Y 346.285,Z 835.208,A -85,B 0,C 180,E1 -13896.055,E2 -13896.055} C_VEL
LIN {X 0,Y 346.063,Z 836.989,A -85,B 0,C 180,E1 -13897.626,E2 -13897.626} C_VEL
LIN {X 0,Y 345.89,Z 838.144,A -85,B 0,C 180,E1 -13899.458,E2 -13899.458} C_VEL
LIN {X 0,Y 345.829,Z 838.305,A -85,B 0,C 180,E1 -13901.244,E2 -13901.244} C_VEL
LIN {X 0,Y 345.86,Z 837.548,A -85,B 0,C 180,E1 -13902.986,E2 -13902.986} C_VEL
LIN {X 0,Y 346.07,Z 835.15,A -85,B 0,C 180,E1 -13905.298,E2 -13905.298} C_VEL
LIN {X 0,Y 346.474,Z 831.3,A -85,B 0,C 180,E1 -13907.468,E2 -13907.468} C_VEL
LIN {X 0,Y 346.951,Z 825.97,A -85,B 0,C 180,E1 -13909.595,E2 -13909.595} C_VEL
LIN {X 0,Y 347.662,Z 819.095,A -85,B 0,C 180,E1 -13911.631,E2 -13911.631} C_VEL
LIN {X 0,Y 348.385,Z 812.091,A -85,B 0,C 180,E1 -13913.279,E2 -13913.279} C_VEL
LIN {X 0,Y 349.398,Z 803.432,A -85,B 0,C 180,E1 -13914.923,E2 -13914.923} C_VEL
LIN {X 0,Y 350.363,Z 794.154,A -85,B 0,C 180,E1 -13916.35,E2 -13916.35} C_VEL
LIN {X 0,Y 351.443,Z 783.665,A -85,B 0,C 180,E1 -13917.662,E2 -13917.662} C_VEL
LIN {X 0,Y 352.487,Z 772.468,A -85,B 0,C 180,E1 -13918.776,E2 -13918.776} C_VEL
LIN {X 0,Y 353.572,Z 759.586,A -85,B 0,C 180,E1 -13919.759,E2 -13919.759} C_VEL
LIN {X 0,Y 352.543,Z 750.228,A -85,B 0,C 180,E1 -13920.391,E2 -13920.391} C_VEL
LIN {X 0,Y 350.29,Z 737.349,A -85,B 0,C 180,E1 -13921.099,E2 -13921.099} C_VEL
LIN {X 0,Y 348.701,Z 729.11,A -85,B 0,C 180,E1 -13921.443,E2 -13921.443} C_VEL
LIN {X 0,Y 349.335,Z 718.624,A -85,B 0,C 180,E1 -13924.866,E2 -13924.866} C_VEL
LIN {X 0,Y 349.963,Z 708.492,A -85,B 0,C 180,E1 -13928.191,E2 -13928.191} C_VEL
LIN {X 0,Y 350.596,Z 697.187,A -85,B 0,C 180,E1 -13931.899,E2 -13931.899} C_VEL
LIN {X 0,Y 351.239,Z 686.185,A -85,B 0,C 180,E1 -13935.516,E2 -13935.516} C_VEL
LIN {X 0,Y 351.501,Z 677.416,A -85,B 0,C 180,E1 -13938.441,E2 -13938.441} C_VEL
LIN {X 0,Y 350.646,Z 670.727,A -85,B 0,C 180,E1 -13940.774,E2 -13940.774} C_VEL
LIN {X 0,Y 349.221,Z 662.669,A -85,B 0,C 180,E1 -13943.646,E2 -13943.646} C_VEL
LIN {X 0,Y 347.902,Z 657.154,A -85,B 0,C 180,E1 -13945.729,E2 -13945.729} C_VEL
LIN {X 0,Y 348.21,Z 657.114,A -85,B 0,C 180,E1 -13947.687,E2 -13947.687} C_VEL
LIN {X 0,Y 348.347,Z 657.096,A -85,B 0,C 180,E1 -13950.001,E2 -13950.001} C_VEL
LIN {X 0,Y 348.21,Z 657.112,A -85,B 0,C 180,E1 -13952.314,E2 -13952.314} C_VEL
LIN {X 0,Y 348.094,Z 657.122,A -85,B 0,C 180,E1 -13956.958,E2 -13956.958} C_VEL
LIN {X 0,Y 347.935,Z 657.143,A -85,B 0,C 180,E1 -13960.475,E2 -13960.475} C_VEL
LIN {X 0,Y 347.9,Z 657.15,A -85,B 0,C 180,E1 -13964.15,E2 -13964.15} C_VEL
LIN {X 0,Y 347.894,Z 657.153,A -85,B 0,C 180,E1 -13968.292,E2 -13968.292} C_VEL
LIN {X 0,Y 347.869,Z 657.156,A -85,B 0,C 180,E1 -13968.585,E2 -13968.585} C_VEL
LIN {X 0,Y 351.715,Z 669.694,A -85,B 0,C 180,E1 -13969.692,E2 -13969.692} C_VEL
LIN {X 0,Y 354.153,Z 678.51,A -85,B 0,C 180,E1 -13970.625,E2 -13970.625} C_VEL
LIN {X 0,Y 353.409,Z 688.715,A -85,B 0,C 180,E1 -13971.694,E2 -13971.694} C_VEL
LIN {X 0,Y 352.524,Z 699.295,A -85,B 0,C 180,E1 -13973.076,E2 -13973.076} C_VEL
LIN {X 0,Y 351.657,Z 708.171,A -85,B 0,C 180,E1 -13974.501,E2 -13974.501} C_VEL
LIN {X 0,Y 350.716,Z 716.631,A -85,B 0,C 180,E1 -13976.159,E2 -13976.159} C_VEL
LIN {X 0,Y 349.928,Z 723.769,A -85,B 0,C 180,E1 -13977.908,E2 -13977.908} C_VEL
LIN {X 0,Y 349.321,Z 728.894,A -85,B 0,C 180,E1 -13979.453,E2 -13979.453} C_VEL
LIN {X 0,Y 348.755,Z 734.371,A -85,B 0,C 180,E1 -13981.598,E2 -13981.598} C_VEL
LIN {X 0,Y 348.435,Z 736.868,A -85,B 0,C 180,E1 -13982.869,E2 -13982.869} C_VEL
LIN {X 0,Y 347.598,Z 738.504,A -85,B 0,C 180,E1 -13983.792,E2 -13983.792} C_VEL
LIN {X 0,Y 344.527,Z 740.729,A -85,B 0,C 180,E1 -13985.308,E2 -13985.308} C_VEL
LIN {X 0,Y 341.565,Z 742.337,A -85,B 0,C 180,E1 -13986.871,E2 -13986.871} C_VEL
LIN {X 0,Y 340.917,Z 742.748,A -85,B 0,C 180,E1 -13987.855,E2 -13987.855} C_VEL
LIN {X 0,Y 341.091,Z 742.77,A -85,B 0,C 180,E1 -13989.698,E2 -13989.698} C_VEL
LIN {X 0,Y 341.282,Z 742.066,A -85,B 0,C 180,E1 -13991.222,E2 -13991.222} C_VEL
LIN {X 0,Y 341.576,Z 740.63,A -85,B 0,C 180,E1 -13992.765,E2 -13992.765} C_VEL
LIN {X 0,Y 342.043,Z 738.482,A -85,B 0,C 180,E1 -13994.315,E2 -13994.315} C_VEL
LIN {X 0,Y 342.593,Z 735.546,A -85,B 0,C 180,E1 -13995.89,E2 -13995.89} C_VEL
LIN {X 0,Y 343.411,Z 730.548,A -85,B 0,C 180,E1 -13997.89,E2 -13997.89} C_VEL
LIN {X 0,Y 344.497,Z 723.92,A -85,B 0,C 180,E1 -13999.909,E2 -13999.909} C_VEL
LIN {X 0,Y 345.637,Z 716.479,A -85,B 0,C 180,E1 -14001.672,E2 -14001.672} C_VEL
LIN {X 0,Y 346.744,Z 708.056,A -85,B 0,C 180,E1 -14003.28,E2 -14003.28} C_VEL
LIN {X 0,Y 347.946,Z 698.978,A -85,B 0,C 180,E1 -14004.677,E2 -14004.677} C_VEL
LIN {X 0,Y 349.061,Z 688.288,A -85,B 0,C 180,E1 -14006.01,E2 -14006.01} C_VEL
LIN {X 0,Y 349.295,Z 683.028,A -85,B 0,C 180,E1 -14006.578,E2 -14006.578} C_VEL
LIN {X 0,Y 345.756,Z 671.3,A -85,B 0,C 180,E1 -14007.959,E2 -14007.959} C_VEL
LIN {X 0,Y 341.691,Z 660.793,A -85,B 0,C 180,E1 -14009.056,E2 -14009.056} C_VEL
LIN {X 0,Y 340.724,Z 658.049,A -85,B 0,C 180,E1 -14009.327,E2 -14009.327} C_VEL
LIN {X 0,Y 340.805,Z 658.03,A -85,B 0,C 180,E1 -14013.02,E2 -14013.02} C_VEL
LIN {X 0,Y 340.756,Z 658.039,A -85,B 0,C 180,E1 -14015.638,E2 -14015.638} C_VEL
LIN {X 0,Y 340.742,Z 658.045,A -85,B 0,C 180,E1 -14019.474,E2 -14019.474} C_VEL
LIN {X 0,Y 340.86,Z 658.029,A -85,B 0,C 180,E1 -14021.985,E2 -14021.985} C_VEL
LIN {X 0,Y 340.871,Z 658.024,A -85,B 0,C 180,E1 -14025.705,E2 -14025.705} C_VEL
LIN {X 0,Y 340.872,Z 658.019,A -85,B 0,C 180,E1 -14029.306,E2 -14029.306} C_VEL
LIN {X 0,Y 341.077,Z 657.991,A -85,B 0,C 180,E1 -14032.898,E2 -14032.898} C_VEL
LIN {X 0,Y 341.171,Z 657.98,A -85,B 0,C 180,E1 -14037.639,E2 -14037.639} C_VEL
LIN {X 0,Y 341.298,Z 657.966,A -85,B 0,C 180,E1 -14040,E2 -14040} C_VEL
LIN {X 0,Y 341.172,Z 657.986,A -85,B 0,C 180,E1 -14042.361,E2 -14042.361} C_VEL
LIN {X 0,Y 341.078,Z 657.997,A -85,B 0,C 180,E1 -14047.102,E2 -14047.102} C_VEL
LIN {X 0,Y 340.873,Z 658.025,A -85,B 0,C 180,E1 -14050.694,E2 -14050.694} C_VEL
LIN {X 0,Y 340.865,Z 658.025,A -85,B 0,C 180,E1 -14054.325,E2 -14054.325} C_VEL
LIN {X 0,Y 340.84,Z 658.029,A -85,B 0,C 180,E1 -14058.467,E2 -14058.467} C_VEL
LIN {X 0,Y 340.756,Z 658.039,A -85,B 0,C 180,E1 -14061.857,E2 -14061.857} C_VEL
LIN {X 0,Y 340.775,Z 658.033,A -85,B 0,C 180,E1 -14065.664,E2 -14065.664} C_VEL
LIN {X 0,Y 340.731,Z 658.04,A -85,B 0,C 180,E1 -14068.321,E2 -14068.321} C_VEL
LIN {X 0,Y 340.7,Z 658.046,A -85,B 0,C 180,E1 -14071.045,E2 -14071.045} C_VEL
LIN {X 0,Y 340.72,Z 658.047,A -85,B 0,C 180,E1 -14075.279,E2 -14075.279} C_VEL
LIN {X 0,Y 340.712,Z 658.047,A -85,B 0,C 180,E1 -14078.386,E2 -14078.386} C_VEL
LIN {X 0,Y 340.756,Z 658.241,A -85,B 0,C 180,E1 -14081.946,E2 -14081.946} C_VEL
LIN {X 0,Y 342.37,Z 665.904,A -85,B 0,C 180,E1 -14085.738,E2 -14085.738} C_VEL
LIN {X 0,Y 343.867,Z 673.499,A -85,B 0,C 180,E1 -14089.154,E2 -14089.154} C_VEL
LIN {X 0,Y 344.849,Z 679.293,A -85,B 0,C 180,E1 -14091.584,E2 -14091.584} C_VEL
LIN {X 0,Y 344.938,Z 681.956,A -85,B 0,C 180,E1 -14092.619,E2 -14092.619} C_VEL
LIN {X 0,Y 343.584,Z 692.578,A -85,B 0,C 180,E1 -14096.476,E2 -14096.476} C_VEL
LIN {X 0,Y 342.471,Z 702.629,A -85,B 0,C 180,E1 -14099.983,E2 -14099.983} C_VEL
LIN {X 0,Y 341.478,Z 713.683,A -85,B 0,C 180,E1 -14103.736,E2 -14103.736} C_VEL
LIN {X 0,Y 340.76,Z 723.357,A -85,B 0,C 180,E1 -14106.929,E2 -14106.929} C_VEL
LIN {X 0,Y 340.573,Z 726.84,A -85,B 0,C 180,E1 -14108.016,E2 -14108.016} C_VEL
LIN {X 0,Y 342.895,Z 741.252,A -85,B 0,C 180,E1 -14108.715,E2 -14108.715} C_VEL
LIN {X 0,Y 344.144,Z 754.363,A -85,B 0,C 180,E1 -14109.529,E2 -14109.529} C_VEL
LIN {X 0,Y 344.597,Z 763.526,A -85,B 0,C 180,E1 -14110.171,E2 -14110.171} C_VEL
LIN {X 0,Y 345.151,Z 776.159,A -85,B 0,C 180,E1 -14110.884,E2 -14110.884} C_VEL
LIN {X 0,Y 345.416,Z 786.046,A -85,B 0,C 180,E1 -14111.616,E2 -14111.616} C_VEL
LIN {X 0,Y 344.365,Z 797.576,A -85,B 0,C 180,E1 -14112.633,E2 -14112.633} C_VEL
LIN {X 0,Y 343.303,Z 808.348,A -85,B 0,C 180,E1 -14113.849,E2 -14113.849} C_VEL
LIN {X 0,Y 342.389,Z 817.765,A -85,B 0,C 180,E1 -14115.164,E2 -14115.164} C_VEL
LIN {X 0,Y 341.497,Z 826.297,A -85,B 0,C 180,E1 -14116.613,E2 -14116.613} C_VEL
LIN {X 0,Y 340.497,Z 834.742,A -85,B 0,C 180,E1 -14118.39,E2 -14118.39} C_VEL
LIN {X 0,Y 339.9,Z 841.512,A -85,B 0,C 180,E1 -14120.178,E2 -14120.178} C_VEL
LIN {X 0,Y 339.471,Z 847.687,A -85,B 0,C 180,E1 -14122.266,E2 -14122.266} C_VEL
LIN {X 0,Y 339.218,Z 852.197,A -85,B 0,C 180,E1 -14124.356,E2 -14124.356} C_VEL
LIN {X 0,Y 339.143,Z 855.279,A -85,B 0,C 180,E1 -14126.435,E2 -14126.435} C_VEL
LIN {X 0,Y 339.099,Z 856.452,A -85,B 0,C 180,E1 -14127.624,E2 -14127.624} C_VEL
LIN {X 0,Y 339.157,Z 857.166,A -85,B 0,C 180,E1 -14128.812,E2 -14128.812} C_VEL
LIN {X 0,Y 339.206,Z 857.479,A -85,B 0,C 180,E1 -14129.999,E2 -14129.999} C_VEL
LIN {X 0,Y 339.14,Z 857.392,A -85,B 0,C 180,E1 -14131.187,E2 -14131.187} C_VEL
LIN {X 0,Y 339.094,Z 856.875,A -85,B 0,C 180,E1 -14132.375,E2 -14132.375} C_VEL
LIN {X 0,Y 339.137,Z 855.929,A -85,B 0,C 180,E1 -14133.564,E2 -14133.564} C_VEL
LIN {X 0,Y 339.174,Z 854.581,A -85,B 0,C 180,E1 -14134.754,E2 -14134.754} C_VEL
LIN {X 0,Y 339.257,Z 851.734,A -85,B 0,C 180,E1 -14136.541,E2 -14136.541} C_VEL
LIN {X 0,Y 339.588,Z 847.844,A -85,B 0,C 180,E1 -14138.329,E2 -14138.329} C_VEL
LIN {X 0,Y 340.075,Z 842.805,A -85,B 0,C 180,E1 -14140.116,E2 -14140.116} C_VEL
LIN {X 0,Y 340.748,Z 836.473,A -85,B 0,C 180,E1 -14141.902,E2 -14141.902} C_VEL
LIN {X 0,Y 341.834,Z 828.551,A -85,B 0,C 180,E1 -14143.676,E2 -14143.676} C_VEL
LIN {X 0,Y 343.032,Z 818.729,A -85,B 0,C 180,E1 -14145.446,E2 -14145.446} C_VEL
LIN {X 0,Y 344.31,Z 808.508,A -85,B 0,C 180,E1 -14146.909,E2 -14146.909} C_VEL
LIN {X 0,Y 345.763,Z 797.072,A -85,B 0,C 180,E1 -14148.21,E2 -14148.21} C_VEL
LIN {X 0,Y 346.899,Z 785.849,A -85,B 0,C 180,E1 -14149.22,E2 -14149.22} C_VEL
LIN {X 0,Y 346.62,Z 773.434,A -85,B 0,C 180,E1 -14150.162,E2 -14150.162} C_VEL
LIN {X 0,Y 346.043,Z 760.256,A -85,B 0,C 180,E1 -14150.92,E2 -14150.92} C_VEL
LIN {X 0,Y 344.481,Z 748.025,A -85,B 0,C 180,E1 -14151.467,E2 -14151.467} C_VEL
LIN {X 0,Y 342.456,Z 737.728,A -85,B 0,C 180,E1 -14151.952,E2 -14151.952} C_VEL
LIN {X 0,Y 340.912,Z 723.348,A -85,B 0,C 180,E1 -14153.461,E2 -14153.461} C_VEL
LIN {X 0,Y 341.727,Z 713.025,A -85,B 0,C 180,E1 -14156.9,E2 -14156.9} C_VEL
LIN {X 0,Y 342.762,Z 702.27,A -85,B 0,C 180,E1 -14160.551,E2 -14160.551} C_VEL
LIN {X 0,Y 343.973,Z 691.745,A -85,B 0,C 180,E1 -14164.185,E2 -14164.185} C_VEL
LIN {X 0,Y 345.105,Z 682.62,A -85,B 0,C 180,E1 -14167.417,E2 -14167.417} C_VEL
LIN {X 0,Y 344.865,Z 678.922,A -85,B 0,C 180,E1 -14168.803,E2 -14168.803} C_VEL
LIN {X 0,Y 343.464,Z 671.669,A -85,B 0,C 180,E1 -14171.68,E2 -14171.68} C_VEL
LIN {X 0,Y 341.588,Z 662.285,A -85,B 0,C 180,E1 -14175.61,E2 -14175.61} C_VEL
LIN {X 0,Y 340.749,Z 658.041,A -85,B 0,C 180,E1 -14177.519,E2 -14177.519} C_VEL
LIN {X 0,Y 340.732,Z 658.044,A -85,B 0,C 180,E1 -14180.252,E2 -14180.252} C_VEL
LIN {X 0,Y 340.707,Z 658.044,A -85,B 0,C 180,E1 -14183.558,E2 -14183.558} C_VEL
LIN {X 0,Y 340.688,Z 658.043,A -85,B 0,C 180,E1 -14186.153,E2 -14186.153} C_VEL
LIN {X 0,Y 340.771,Z 658.035,A -85,B 0,C 180,E1 -14190.332,E2 -14190.332} C_VEL
LIN {X 0,Y 340.801,Z 658.034,A -85,B 0,C 180,E1 -14193.019,E2 -14193.019} C_VEL
LIN {X 0,Y 340.724,Z 658.038,A -85,B 0,C 180,E1 -14196.927,E2 -14196.927} C_VEL
LIN {X 0,Y 340.79,Z 658.033,A -85,B 0,C 180,E1 -14200.733,E2 -14200.733} C_VEL
LIN {X 0,Y 340.782,Z 658.035,A -85,B 0,C 180,E1 -14203.218,E2 -14203.218} C_VEL
LIN {X 0,Y 340.842,Z 658.026,A -85,B 0,C 180,E1 -14206.89,E2 -14206.89} C_VEL
LIN {X 0,Y 340.925,Z 658.019,A -85,B 0,C 180,E1 -14210.507,E2 -14210.507} C_VEL
LIN {X 0,Y 341.07,Z 658,A -85,B 0,C 180,E1 -14212.898,E2 -14212.898} C_VEL
LIN {X 0,Y 341.043,Z 658.165,A -85,B 0,C 180,E1 -14214.234,E2 -14214.234} C_VEL
LIN {X 0,Y 343.761,Z 668.203,A -85,B 0,C 180,E1 -14218.242,E2 -14218.242} C_VEL
LIN {X 0,Y 345.018,Z 674.435,A -85,B 0,C 180,E1 -14220.583,E2 -14220.583} C_VEL
LIN {X 0,Y 345.694,Z 679.279,A -85,B 0,C 180,E1 -14222.33,E2 -14222.33} C_VEL
LIN {X 0,Y 345.661,Z 686.106,A -85,B 0,C 180,E1 -14224.665,E2 -14224.665} C_VEL
LIN {X 0,Y 344.957,Z 695.008,A -85,B 0,C 180,E1 -14227.61,E2 -14227.61} C_VEL
LIN {X 0,Y 344.216,Z 706.845,A -85,B 0,C 180,E1 -14231.474,E2 -14231.474} C_VEL
LIN {X 0,Y 343.44,Z 716.994,A -85,B 0,C 180,E1 -14234.82,E2 -14234.82} C_VEL
LIN {X 0,Y 342.813,Z 726.341,A -85,B 0,C 180,E1 -14237.909,E2 -14237.909} C_VEL
LIN {X 0,Y 342.615,Z 729.988,A -85,B 0,C 180,E1 -14239.117,E2 -14239.117} C_VEL
LIN {X 0,Y 346.222,Z 744.789,A -85,B 0,C 180,E1 -14239.993,E2 -14239.993} C_VEL
LIN {X 0,Y 348.131,Z 756.679,A -85,B 0,C 180,E1 -14240.83,E2 -14240.83} C_VEL
LIN {X 0,Y 348.46,Z 761.625,A -85,B 0,C 180,E1 -14241.208,E2 -14241.208} C_VEL
LIN {X 0,Y 347.221,Z 774.36,A -85,B 0,C 180,E1 -14242.233,E2 -14242.233} C_VEL
LIN {X 0,Y 345.812,Z 786.229,A -85,B 0,C 180,E1 -14243.486,E2 -14243.486} C_VEL
LIN {X 0,Y 344.477,Z 796.743,A -85,B 0,C 180,E1 -14244.884,E2 -14244.884} C_VEL
LIN {X 0,Y 343.356,Z 805.143,A -85,B 0,C 180,E1 -14246.265,E2 -14246.265} C_VEL
LIN {X 0,Y 342.146,Z 813.57,A -85,B 0,C 180,E1 -14247.964,E2 -14247.964} C_VEL
LIN {X 0,Y 341.191,Z 820.278,A -85,B 0,C 180,E1 -14249.628,E2 -14249.628} C_VEL
LIN {X 0,Y 340.425,Z 826.551,A -85,B 0,C 180,E1 -14251.58,E2 -14251.58} C_VEL
LIN {X 0,Y 339.841,Z 830.689,A -85,B 0,C 180,E1 -14253.232,E2 -14253.232} C_VEL
LIN {X 0,Y 339.295,Z 834.764,A -85,B 0,C 180,E1 -14255.449,E2 -14255.449} C_VEL
LIN {X 0,Y 339.058,Z 836.689,A -85,B 0,C 180,E1 -14256.95,E2 -14256.95} C_VEL
LIN {X 0,Y 338.892,Z 837.921,A -85,B 0,C 180,E1 -14258.473,E2 -14258.473} C_VEL
LIN {X 0,Y 338.782,Z 838.517,A -85,B 0,C 180,E1 -14260.023,E2 -14260.023} C_VEL
LIN {X 0,Y 338.738,Z 838.413,A -85,B 0,C 180,E1 -14261.678,E2 -14261.678} C_VEL
LIN {X 0,Y 338.81,Z 837.417,A -85,B 0,C 180,E1 -14263.448,E2 -14263.448} C_VEL
LIN {X 0,Y 339.06,Z 834.669,A -85,B 0,C 180,E1 -14265.787,E2 -14265.787} C_VEL
LIN {X 0,Y 339.413,Z 831.438,A -85,B 0,C 180,E1 -14267.578,E2 -14267.578} C_VEL
LIN {X 0,Y 339.743,Z 827.433,A -85,B 0,C 180,E1 -14269.255,E2 -14269.255} C_VEL
LIN {X 0,Y 340.471,Z 820.986,A -85,B 0,C 180,E1 -14271.339,E2 -14271.339} C_VEL
LIN {X 0,Y 341.142,Z 814.685,A -85,B 0,C 180,E1 -14272.945,E2 -14272.945} C_VEL
LIN {X 0,Y 342.151,Z 806.032,A -85,B 0,C 180,E1 -14274.72,E2 -14274.72} C_VEL
LIN {X 0,Y 343.183,Z 796.788,A -85,B 0,C 180,E1 -14276.257,E2 -14276.257} C_VEL
LIN {X 0,Y 344.269,Z 786.767,A -85,B 0,C 180,E1 -14277.605,E2 -14277.605} C_VEL
LIN {X 0,Y 345.409,Z 774.914,A -85,B 0,C 180,E1 -14278.874,E2 -14278.874} C_VEL
LIN {X 0,Y 346.519,Z 762.884,A -85,B 0,C 180,E1 -14279.87,E2 -14279.87} C_VEL
LIN {X 0,Y 346.643,Z 757.983,A -85,B 0,C 180,E1 -14280.217,E2 -14280.217} C_VEL
LIN {X 0,Y 344.683,Z 744.684,A -85,B 0,C 180,E1 -14281.079,E2 -14281.079} C_VEL
LIN {X 0,Y 342.147,Z 731.342,A -85,B 0,C 180,E1 -14281.725,E2 -14281.725} C_VEL
LIN {X 0,Y 341.755,Z 729.196,A -85,B 0,C 180,E1 -14281.834,E2 -14281.834} C_VEL
LIN {X 0,Y 342.36,Z 719.06,A -85,B 0,C 180,E1 -14285.185,E2 -14285.185} C_VEL
LIN {X 0,Y 343.021,Z 709.474,A -85,B 0,C 180,E1 -14288.36,E2 -14288.36} C_VEL
LIN {X 0,Y 343.673,Z 698.104,A -85,B 0,C 180,E1 -14292.138,E2 -14292.138} C_VEL
LIN {X 0,Y 344.356,Z 687.035,A -85,B 0,C 180,E1 -14295.824,E2 -14295.824} C_VEL
LIN {X 0,Y 344.598,Z 678.755,A -85,B 0,C 180,E1 -14298.623,E2 -14298.623} C_VEL
LIN {X 0,Y 343.63,Z 671.565,A -85,B 0,C 180,E1 -14301.177,E2 -14301.177} C_VEL
LIN {X 0,Y 342.153,Z 663.481,A -85,B 0,C 180,E1 -14304.106,E2 -14304.106} C_VEL
LIN {X 0,Y 340.879,Z 658.029,A -85,B 0,C 180,E1 -14306.159,E2 -14306.159} C_VEL
LIN {X 0,Y 341.171,Z 657.991,A -85,B 0,C 180,E1 -14307.639,E2 -14307.639} C_VEL
LIN {X 0,Y 341.298,Z 657.974,A -85,B 0,C 180,E1 -14310.001,E2 -14310.001} C_VEL
LIN {X 0,Y 341.171,Z 657.989,A -85,B 0,C 180,E1 -14312.362,E2 -14312.362} C_VEL
LIN {X 0,Y 341.062,Z 657.998,A -85,B 0,C 180,E1 -14317.103,E2 -14317.103} C_VEL
LIN {X 0,Y 340.877,Z 658.023,A -85,B 0,C 180,E1 -14320.694,E2 -14320.694} C_VEL
LIN {X 0,Y 340.864,Z 658.026,A -85,B 0,C 180,E1 -14324.325,E2 -14324.325} C_VEL
LIN {X 0,Y 340.859,Z 658.029,A -85,B 0,C 180,E1 -14328.201,E2 -14328.201} C_VEL
LIN {X 0,Y 344.654,Z 670.465,A -85,B 0,C 180,E1 -14329.334,E2 -14329.334} C_VEL
LIN {X 0,Y 347.378,Z 680.536,A -85,B 0,C 180,E1 -14330.426,E2 -14330.426} C_VEL
LIN {X 0,Y 346.383,Z 692.29,A -85,B 0,C 180,E1 -14331.734,E2 -14331.734} C_VEL
LIN {X 0,Y 345.591,Z 701.388,A -85,B 0,C 180,E1 -14332.99,E2 -14332.99} C_VEL
LIN {X 0,Y 344.726,Z 709.768,A -85,B 0,C 180,E1 -14334.384,E2 -14334.384} C_VEL
LIN {X 0,Y 343.812,Z 717.412,A -85,B 0,C 180,E1 -14335.918,E2 -14335.918} C_VEL
LIN {X 0,Y 342.963,Z 724.905,A -85,B 0,C 180,E1 -14337.788,E2 -14337.788} C_VEL
LIN {X 0,Y 342.16,Z 731.599,A -85,B 0,C 180,E1 -14339.935,E2 -14339.935} C_VEL
LIN {X 0,Y 341.726,Z 735.641,A -85,B 0,C 180,E1 -14341.631,E2 -14341.631} C_VEL
LIN {X 0,Y 341.258,Z 739.435,A -85,B 0,C 180,E1 -14343.783,E2 -14343.783} C_VEL
LIN {X 0,Y 341.046,Z 741.173,A -85,B 0,C 180,E1 -14345.24,E2 -14345.24} C_VEL
LIN {X 0,Y 340.93,Z 742.331,A -85,B 0,C 180,E1 -14346.714,E2 -14346.714} C_VEL
LIN {X 0,Y 340.917,Z 742.748,A -85,B 0,C 180,E1 -14347.855,E2 -14347.855} C_VEL
LIN {X 0,Y 340.319,Z 743.048,A -85,B 0,C 180,E1 -14348.842,E2 -14348.842} C_VEL
LIN {X 0,Y 337.646,Z 743.133,A -85,B 0,C 180,E1 -14350.456,E2 -14350.456} C_VEL
LIN {X 0,Y 335.462,Z 742.633,A -85,B 0,C 180,E1 -14351.757,E2 -14351.757} C_VEL
LIN {X 0,Y 334.653,Z 741.836,A -85,B 0,C 180,E1 -14352.751,E2 -14352.751} C_VEL
LIN {X 0,Y 334.657,Z 741.434,A -85,B 0,C 180,E1 -14353.083,E2 -14353.083} C_VEL
LIN {X 0,Y 335.096,Z 739.509,A -85,B 0,C 180,E1 -14354.514,E2 -14354.514} C_VEL
LIN {X 0,Y 335.771,Z 736.143,A -85,B 0,C 180,E1 -14356.313,E2 -14356.313} C_VEL
LIN {X 0,Y 336.507,Z 731.848,A -85,B 0,C 180,E1 -14358.062,E2 -14358.062} C_VEL
LIN {X 0,Y 337.463,Z 726.447,A -85,B 0,C 180,E1 -14359.789,E2 -14359.789} C_VEL
LIN {X 0,Y 338.646,Z 719.186,A -85,B 0,C 180,E1 -14361.637,E2 -14361.637} C_VEL
LIN {X 0,Y 339.703,Z 711.932,A -85,B 0,C 180,E1 -14363.132,E2 -14363.132} C_VEL
LIN {X 0,Y 340.84,Z 703.871,A -85,B 0,C 180,E1 -14364.499,E2 -14364.499} C_VEL
LIN {X 0,Y 342.007,Z 694.221,A -85,B 0,C 180,E1 -14365.842,E2 -14365.842} C_VEL
LIN {X 0,Y 342.806,Z 686.391,A -85,B 0,C 180,E1 -14366.742,E2 -14366.742} C_VEL
LIN {X 0,Y 342.125,Z 682.791,A -85,B 0,C 180,E1 -14367.194,E2 -14367.194} C_VEL
LIN {X 0,Y 338.948,Z 672.638,A -85,B 0,C 180,E1 -14368.429,E2 -14368.429} C_VEL
LIN {X 0,Y 334.832,Z 661.982,A -85,B 0,C 180,E1 -14369.577,E2 -14369.577} C_VEL
LIN {X 0,Y 333.695,Z 658.921,A -85,B 0,C 180,E1 -14369.894,E2 -14369.894} C_VEL
LIN {X 0,Y 333.736,Z 658.907,A -85,B 0,C 180,E1 -14373.754,E2 -14373.754} C_VEL
LIN {X 0,Y 333.661,Z 658.915,A -85,B 0,C 180,E1 -14377.72,E2 -14377.72} C_VEL
LIN {X 0,Y 333.796,Z 658.911,A -85,B 0,C 180,E1 -14381.59,E2 -14381.59} C_VEL
LIN {X 0,Y 333.81,Z 658.904,A -85,B 0,C 180,E1 -14385.577,E2 -14385.577} C_VEL
LIN {X 0,Y 333.835,Z 658.895,A -85,B 0,C 180,E1 -14389.078,E2 -14389.078} C_VEL
LIN {X 0,Y 334.027,Z 658.868,A -85,B 0,C 180,E1 -14392.748,E2 -14392.748} C_VEL
LIN {X 0,Y 333.813,Z 658.902,A -85,B 0,C 180,E1 -14395.169,E2 -14395.169} C_VEL
LIN {X 0,Y 334.109,Z 658.859,A -85,B 0,C 180,E1 -14397.589,E2 -14397.589} C_VEL
LIN {X 0,Y 334.249,Z 658.843,A -85,B 0,C 180,E1 -14400,E2 -14400} C_VEL
LIN {X 0,Y 334.109,Z 658.867,A -85,B 0,C 180,E1 -14402.411,E2 -14402.411} C_VEL
LIN {X 0,Y 334.027,Z 658.875,A -85,B 0,C 180,E1 -14407.253,E2 -14407.253} C_VEL
LIN {X 0,Y 333.836,Z 658.9,A -85,B 0,C 180,E1 -14410.922,E2 -14410.922} C_VEL
LIN {X 0,Y 333.81,Z 658.905,A -85,B 0,C 180,E1 -14414.634,E2 -14414.634} C_VEL
LIN {X 0,Y 333.799,Z 658.904,A -85,B 0,C 180,E1 -14418.655,E2 -14418.655} C_VEL
LIN {X 0,Y 333.695,Z 658.917,A -85,B 0,C 180,E1 -14422.278,E2 -14422.278} C_VEL
LIN {X 0,Y 333.737,Z 658.911,A -85,B 0,C 180,E1 -14426.246,E2 -14426.246} C_VEL
LIN {X 0,Y 333.692,Z 658.92,A -85,B 0,C 180,E1 -14428.974,E2 -14428.974} C_VEL
LIN {X 0,Y 333.646,Z 658.925,A -85,B 0,C 180,E1 -14432.587,E2 -14432.587} C_VEL
LIN {X 0,Y 333.678,Z 658.924,A -85,B 0,C 180,E1 -14436.139,E2 -14436.139} C_VEL
LIN {X 0,Y 333.649,Z 658.929,A -85,B 0,C 180,E1 -14439.192,E2 -14439.192} C_VEL
LIN {X 0,Y 333.681,Z 659.019,A -85,B 0,C 180,E1 -14441.262,E2 -14441.262} C_VEL
LIN {X 0,Y 335.003,Z 665.248,A -85,B 0,C 180,E1 -14444.497,E2 -14444.497} C_VEL
LIN {X 0,Y 336.49,Z 672.771,A -85,B 0,C 180,E1 -14448.059,E2 -14448.059} C_VEL
LIN {X 0,Y 337.878,Z 680.412,A -85,B 0,C 180,E1 -14451.39,E2 -14451.39} C_VEL
LIN {X 0,Y 338.047,Z 682.386,A -85,B 0,C 180,E1 -14452.188,E2 -14452.188} C_VEL
LIN {X 0,Y 336.801,Z 691.757,A -85,B 0,C 180,E1 -14455.708,E2 -14455.708} C_VEL
LIN {X 0,Y 335.463,Z 703.19,A -85,B 0,C 180,E1 -14459.814,E2 -14459.814} C_VEL
LIN {X 0,Y 334.549,Z 712.797,A -85,B 0,C 180,E1 -14463.149,E2 -14463.149} C_VEL
LIN {X 0,Y 333.658,Z 724.34,A -85,B 0,C 180,E1 -14467.066,E2 -14467.066} C_VEL
LIN {X 0,Y 333.571,Z 725.494,A -85,B 0,C 180,E1 -14467.448,E2 -14467.448} C_VEL
LIN {X 0,Y 335.97,Z 739.801,A -85,B 0,C 180,E1 -14468.168,E2 -14468.168} C_VEL
LIN {X 0,Y 337.274,Z 752.477,A -85,B 0,C 180,E1 -14468.976,E2 -14468.976} C_VEL
LIN {X 0,Y 337.813,Z 764.507,A -85,B 0,C 180,E1 -14469.873,E2 -14469.873} C_VEL
LIN {X 0,Y 338.308,Z 777.69,A -85,B 0,C 180,E1 -14470.665,E2 -14470.665} C_VEL
LIN {X 0,Y 338.493,Z 786.976,A -85,B 0,C 180,E1 -14471.383,E2 -14471.383} C_VEL
LIN {X 0,Y 337.39,Z 798.204,A -85,B 0,C 180,E1 -14472.419,E2 -14472.419} C_VEL
LIN {X 0,Y 336.363,Z 808.486,A -85,B 0,C 180,E1 -14473.616,E2 -14473.616} C_VEL
LIN {X 0,Y 335.433,Z 817.66,A -85,B 0,C 180,E1 -14474.927,E2 -14474.927} C_VEL
LIN {X 0,Y 334.535,Z 825.765,A -85,B 0,C 180,E1 -14476.329,E2 -14476.329} C_VEL
LIN {X 0,Y 333.652,Z 833.008,A -85,B 0,C 180,E1 -14477.84,E2 -14477.84} C_VEL
LIN {X 0,Y 332.95,Z 840.095,A -85,B 0,C 180,E1 -14479.663,E2 -14479.663} C_VEL
LIN {X 0,Y 332.504,Z 845.722,A -85,B 0,C 180,E1 -14481.491,E2 -14481.491} C_VEL
LIN {X 0,Y 332.217,Z 850.113,A -85,B 0,C 180,E1 -14483.318,E2 -14483.318} C_VEL
LIN {X 0,Y 332.106,Z 853.393,A -85,B 0,C 180,E1 -14485.144,E2 -14485.144} C_VEL
LIN {X 0,Y 332.069,Z 855.008,A -85,B 0,C 180,E1 -14486.359,E2 -14486.359} C_VEL
LIN {X 0,Y 332.012,Z 856.204,A -85,B 0,C 180,E1 -14487.573,E2 -14487.573} C_VEL
LIN {X 0,Y 332.057,Z 856.941,A -85,B 0,C 180,E1 -14488.787,E2 -14488.787} C_VEL
LIN {X 0,Y 332.108,Z 857.27,A -85,B 0,C 180,E1 -14489.999,E2 -14489.999} C_VEL
LIN {X 0,Y 332.04,Z 857.197,A -85,B 0,C 180,E1 -14491.212,E2 -14491.212} C_VEL
LIN {X 0,Y 332.007,Z 856.711,A -85,B 0,C 180,E1 -14492.426,E2 -14492.426} C_VEL
LIN {X 0,Y 332.062,Z 855.78,A -85,B 0,C 180,E1 -14493.64,E2 -14493.64} C_VEL
LIN {X 0,Y 332.122,Z 852.848,A -85,B 0,C 180,E1 -14495.975,E2 -14495.975} C_VEL
LIN {X 0,Y 332.39,Z 849.199,A -85,B 0,C 180,E1 -14497.899,E2 -14497.899} C_VEL
LIN {X 0,Y 332.862,Z 844.59,A -85,B 0,C 180,E1 -14499.724,E2 -14499.724} C_VEL
LIN {X 0,Y 333.636,Z 837.607,A -85,B 0,C 180,E1 -14501.851,E2 -14501.851} C_VEL
LIN {X 0,Y 334.757,Z 830.083,A -85,B 0,C 180,E1 -14503.661,E2 -14503.661} C_VEL
LIN {X 0,Y 335.762,Z 822.428,A -85,B 0,C 180,E1 -14505.167,E2 -14505.167} C_VEL
LIN {X 0,Y 337.02,Z 813.119,A -85,B 0,C 180,E1 -14506.661,E2 -14506.661} C_VEL
LIN {X 0,Y 338.345,Z 802.842,A -85,B 0,C 180,E1 -14507.997,E2 -14507.997} C_VEL
LIN {X 0,Y 339.791,Z 791.527,A -85,B 0,C 180,E1 -14509.168,E2 -14509.168} C_VEL
LIN {X 0,Y 340.193,Z 784.646,A -85,B 0,C 180,E1 -14509.772,E2 -14509.772} C_VEL
LIN {X 0,Y 340.019,Z 772.614,A -85,B 0,C 180,E1 -14510.687,E2 -14510.687} C_VEL
LIN {X 0,Y 339.432,Z 759.569,A -85,B 0,C 180,E1 -14511.455,E2 -14511.455} C_VEL
LIN {X 0,Y 337.879,Z 748.192,A -85,B 0,C 180,E1 -14511.995,E2 -14511.995} C_VEL
LIN {X 0,Y 335.819,Z 737.801,A -85,B 0,C 180,E1 -14512.496,E2 -14512.496} C_VEL
LIN {X 0,Y 334.032,Z 721.171,A -85,B 0,C 180,E1 -14514.345,E2 -14514.345} C_VEL
LIN {X 0,Y 335.056,Z 709.787,A -85,B 0,C 180,E1 -14518.239,E2 -14518.239} C_VEL
LIN {X 0,Y 336.254,Z 698.459,A -85,B 0,C 180,E1 -14522.205,E2 -14522.205} C_VEL
LIN {X 0,Y 337.761,Z 686.809,A -85,B 0,C 180,E1 -14526.37,E2 -14526.37} C_VEL
LIN {X 0,Y 338.145,Z 682.826,A -85,B 0,C 180,E1 -14527.834,E2 -14527.834} C_VEL
LIN {X 0,Y 337.523,Z 678.303,A -85,B 0,C 180,E1 -14529.608,E2 -14529.608} C_VEL
LIN {X 0,Y 335.948,Z 670.206,A -85,B 0,C 180,E1 -14532.929,E2 -14532.929} C_VEL
LIN {X 0,Y 334.488,Z 662.873,A -85,B 0,C 180,E1 -14536.102,E2 -14536.102} C_VEL
LIN {X 0,Y 333.717,Z 658.918,A -85,B 0,C 180,E1 -14537.935,E2 -14537.935} C_VEL
LIN {X 0,Y 333.679,Z 658.921,A -85,B 0,C 180,E1 -14541.195,E2 -14541.195} C_VEL
LIN {X 0,Y 333.682,Z 658.913,A -85,B 0,C 180,E1 -14545.225,E2 -14545.225} C_VEL
LIN {X 0,Y 333.693,Z 658.918,A -85,B 0,C 180,E1 -14549.637,E2 -14549.637} C_VEL
LIN {X 0,Y 333.74,Z 658.913,A -85,B 0,C 180,E1 -14552.401,E2 -14552.401} C_VEL
LIN {X 0,Y 333.722,Z 658.912,A -85,B 0,C 180,E1 -14555.09,E2 -14555.09} C_VEL
LIN {X 0,Y 333.682,Z 658.919,A -85,B 0,C 180,E1 -14559.019,E2 -14559.019} C_VEL
LIN {X 0,Y 333.79,Z 658.906,A -85,B 0,C 180,E1 -14561.589,E2 -14561.589} C_VEL
LIN {X 0,Y 333.803,Z 658.905,A -85,B 0,C 180,E1 -14565.576,E2 -14565.576} C_VEL
LIN {X 0,Y 333.833,Z 658.899,A -85,B 0,C 180,E1 -14569.078,E2 -14569.078} C_VEL
LIN {X 0,Y 334.02,Z 658.878,A -85,B 0,C 180,E1 -14572.747,E2 -14572.747} C_VEL
LIN {X 0,Y 334.027,Z 658.953,A -85,B 0,C 180,E1 -14573.203,E2 -14573.203} C_VEL
LIN {X 0,Y 336.944,Z 669.551,A -85,B 0,C 180,E1 -14577.609,E2 -14577.609} C_VEL
LIN {X 0,Y 338.226,Z 675.684,A -85,B 0,C 180,E1 -14580,E2 -14580} C_VEL
LIN {X 0,Y 339.057,Z 682.089,A -85,B 0,C 180,E1 -14582.376,E2 -14582.376} C_VEL
LIN {X 0,Y 338.943,Z 688.007,A -85,B 0,C 180,E1 -14584.456,E2 -14584.456} C_VEL
LIN {X 0,Y 338.151,Z 697.979,A -85,B 0,C 180,E1 -14587.764,E2 -14587.764} C_VEL
LIN {X 0,Y 337.307,Z 709.707,A -85,B 0,C 180,E1 -14591.691,E2 -14591.691} C_VEL
LIN {X 0,Y 336.49,Z 719.986,A -85,B 0,C 180,E1 -14595.134,E2 -14595.134} C_VEL
LIN {X 0,Y 335.79,Z 730.202,A -85,B 0,C 180,E1 -14598.564,E2 -14598.564} C_VEL
LIN {X 0,Y 339.382,Z 744.331,A -85,B 0,C 180,E1 -14599.423,E2 -14599.423} C_VEL
LIN {X 0,Y 341.383,Z 756.768,A -85,B 0,C 180,E1 -14600.328,E2 -14600.328} C_VEL
LIN {X 0,Y 341.937,Z 761.54,A -85,B 0,C 180,E1 -14600.722,E2 -14600.722} C_VEL
LIN {X 0,Y 340.776,Z 773.283,A -85,B 0,C 180,E1 -14601.67,E2 -14601.67} C_VEL
LIN {X 0,Y 339.415,Z 784.625,A -85,B 0,C 180,E1 -14602.845,E2 -14602.845} C_VEL
LIN {X 0,Y 338.049,Z 794.981,A -85,B 0,C 180,E1 -14604.2,E2 -14604.2} C_VEL
LIN {X 0,Y 336.717,Z 804.093,A -85,B 0,C 180,E1 -14605.664,E2 -14605.664} C_VEL
LIN {X 0,Y 335.43,Z 813.005,A -85,B 0,C 180,E1 -14607.448,E2 -14607.448} C_VEL
LIN {X 0,Y 334.331,Z 820.213,A -85,B 0,C 180,E1 -14609.25,E2 -14609.25} C_VEL
LIN {X 0,Y 333.529,Z 826.066,A -85,B 0,C 180,E1 -14611.081,E2 -14611.081} C_VEL
LIN {X 0,Y 332.748,Z 831.516,A -85,B 0,C 180,E1 -14613.308,E2 -14613.308} C_VEL
LIN {X 0,Y 332.196,Z 835.404,A -85,B 0,C 180,E1 -14615.577,E2 -14615.577} C_VEL
